// TwinCAT 3 PLC project TAMAR_22mm
// ProgramVersion: 3.1.4023.0
// libraries:
//   Tc2_MC2, * (Beckhoff Automation GmbH)
//   Tc2_Standard, * (Beckhoff Automation GmbH)
//   Tc2_System, * (Beckhoff Automation GmbH)
//   Tc2_Utilities, * (Beckhoff Automation GmbH)
//   Tc3_Module, * (Beckhoff Automation GmbH)
//   VisuDialogs, * (System)
// project tree:
//   Checks/ CheckBounds.TcPOU, CheckDivDInt.TcPOU, CheckDivLInt.TcPOU, CheckDivLReal.TcPOU, CheckDivReal.TcPOU, CheckLRangeSigned.TcPOU, CheckLRangeUnsigned.TcPOU, CheckPointer.TcPOU, CheckRangeSigned.TcPOU, CheckRangeUnsigned.TcPOU
//   DUTs/ ePistonStatus.TcDUT, E_CONVAYOR_STATE.TcDUT, E_EventType.TcDUT (not stored), E_MAIN_STATE.TcDUT, E_PISTON_STATE.TcDUT (not stored), E_PISTON_TYPE.TcDUT (not stored), E_STATION_STATE.TcDUT, ST_CART.TcDUT, ST_CsvTableRowData.TcDUT, ST_Event.TcDUT, ST_PISTON.TcDUT
//   Functions/ F_Linear.TcPOU, UpdateEventTimestampWithSystemTime.TcPOU, UpdateTimeStamp.TcPOU
//   / GlobalTextList.TcGTLO, PlcTask.TcTTO (not stored), Visualization Manager.TcVMO (not stored)
//   GVLs/ GVL.TcGVL, GVL_EVENT_LOGS.TcGVL
//   IO/ EL1809.TcDUT (not stored), EL2869.TcDUT, GVL_IO.TcGVL, ST_VTUG.TcDUT (not stored)
//   POUs/AXES/ FB_Axis.TcPOU
//   POUs/ FB_CART.TcPOU, FB_ERROR_CODE.TcPOU, FB_EventLogger.TcPOU, FB_PISTON.TcPOU, MAIN.TcPOU, MOTORS.TcPOU, PISTONS_CYCLE.TcPOU, prg_CSV_V2.TcPOU
//   POUs/PISTONS/ E_PIST_STATUS.TcDUT, E_PIST_TYPE.TcDUT, FB_PIST.TcPOU, GVL_PIST.TcGVL, PIST_CYCLE.TcPOU
//   STATIONS/ FB_CLEAN.TcPOU, FB_DROP.TcPOU, FB_MAIN_CONV.TcPOU, FB_SEPARATE.TcPOU, FB_STATION.TcPOU, FB_SUPPLY.TcPOU, FB_SUPPLY_CONV.TcPOU, _SEPARATE.TcPOU
// real-time tasks:
//   TASK PlcTask: cycle T#10ms, priority 20, ADS port 350
// motion (NC):
//   TASK NC-Task 1 SAF: cycle T#2ms, priority 4, ADS port 501
//   TASK NC-Task 1 SVB: cycle T#10ms, priority 8, ADS port 511
//   AXIS MAIN (id 1)
//     OtherSettings: AllowMotionCmdToSlave=true
//     encoder EncType=19
//       EncPara: MaxCount=#xffffffff
//     drive DrvType=16
//       DrvPara: MaxCount=#xffffffff, DriveControlDWord=#x00000100
//         Analog: TorqueSetpointScale=10, ScaleFactorActTorque=0.1
//         TimeComp: TaskDelayCycles=1
//     controller CtrType=1
//       CtrPara: PriorControlFactor=1
//         Observer: BandWidth=20
//   AXIS SUPPLY (id 2)
//     OtherSettings: AllowMotionCmdToSlave=true
//     encoder EncType=19
//       EncPara: MaxCount=#xffffffff
//     drive DrvType=16
//       DrvPara: MaxCount=#xffffffff, DriveControlDWord=#x00000100
//         Analog: TorqueSetpointScale=10, ScaleFactorActTorque=0.1
//         TimeComp: TaskDelayCycles=1
//     controller CtrType=1
//       CtrPara: PriorControlFactor=1
//         Observer: BandWidth=20
//   AXIS JACK1 (id 3)
//     OtherSettings: AllowMotionCmdToSlave=true
//     encoder EncType=1
//     drive DrvType=5
//       Analog: TorqueSetpointScale=10, ScaleFactorActTorque=0.1
//       TimeComp: TaskDelayCycles=1
//     controller CtrType=1
//       CtrPara: PriorControlFactor=1
//         Observer: BandWidth=20
//   AXIS JACK2 (id 4)
//     OtherSettings: AllowMotionCmdToSlave=true
//     encoder EncType=1
//     drive DrvType=5
//       Analog: TorqueSetpointScale=10, ScaleFactorActTorque=0.1
//     controller CtrType=1
//       CtrPara: PriorControlFactor=1
//         Observer: BandWidth=20
// I/O:
//   DEVICE Device 3 (EtherCAT), AmsNetId 5.109.70.127.4.1
//     Term 1 (EK1100) [EK1100 EtherCAT Coupler (2A E-Bus)]
//       Term 2 (EL1809) [EL1809 16Ch. Dig. Input 24V, 3ms]
//       Term 10 (EL1809) [EL1809 16Ch. Dig. Input 24V, 3ms]
//       Term 11 (EL1809) [EL1809 16Ch. Dig. Input 24V, 3ms]
//       Term 13 (EL1809) [EL1809 16Ch. Dig. Input 24V, 3ms]
//       Term 3 (EL2869) [EL2869 16Ch. Dig Output 24V, 0.5A, Diagnostic]
//       Term 4 (EL6224) [EL6224 (IO Link Master)]
//       Term 15 (EL9011) [EL9011 End Terminal]
//       Term 7 (EL9011) [EL9011 End Terminal]
//     MAIN
//     SUPPLY [CD02 EtherCAT Drive (CoE)]
// variable links:
//   (this object) <-> Device 3 (EtherCAT)/MAIN
//     Drive/Inputs/In/nDataIn1 <-> TxPDO 1/Following Error Actual Value
//     Drive/Inputs/In/nDataIn3[0] <-> TxPDO 4/Torque Actual Value
//     Drive/Inputs/In/nDcOutputTime <-> InfoData/DcOutputShift
//     Drive/Inputs/In/nState1 <-> TxPDO 4/Statusword
//     Drive/Inputs/In/nState2 <-> TxPDO 4/Statusword @bit 8
//     Drive/Inputs/In/nState4 @bit 1 <-> WcState/InputToggle
//     Drive/Inputs/In/nState4 <-> WcState/WcState
//     Drive/Inputs/In/nState5 <-> TxPDO 3/Modes of Operation Display
//     Drive/Outputs/Out/nCtrl1 <-> RxPDO 4/Controlword
//     Drive/Outputs/Out/nCtrl2 <-> RxPDO 4/Controlword @bit 8
//     Drive/Outputs/Out/nCtrl5 <-> RxPDO 4/Modes of Operation
//     Drive/Outputs/Out/nDataOut1 <-> RxPDO 1/Target Position
//     Drive/Outputs/Out/nDataOut2 <-> RxPDO 2/Target Velocity
//     Drive/Outputs/Out/nDataOut3[0] <-> RxPDO 4/Torque Offset
//     Drive/Outputs/Out/nDataOut4[0] <-> RxPDO 3/Target Torque
//     Enc/Inputs/In/nDataIn1 <-> TxPDO 2/Position Actual Value
//     Enc/Inputs/In/nDcInputTime <-> InfoData/DcInputShift
//     Enc/Inputs/In/nState4 @bit 1 <-> WcState/InputToggle
//     Enc/Inputs/In/nState4 <-> WcState/WcState
//   (this object) <-> Device 3 (EtherCAT)/SUPPLY
//     Drive/Inputs/In/nDataIn1 <-> TxPDO 1/Following Error Actual Value
//     Drive/Inputs/In/nDataIn3[0] <-> TxPDO 4/Torque Actual Value
//     Drive/Inputs/In/nDcOutputTime <-> InfoData/DcOutputShift
//     Drive/Inputs/In/nState1 <-> TxPDO 4/Statusword
//     Drive/Inputs/In/nState2 <-> TxPDO 4/Statusword @bit 8
//     Drive/Inputs/In/nState4 @bit 1 <-> WcState/InputToggle
//     Drive/Inputs/In/nState4 <-> WcState/WcState
//     Drive/Inputs/In/nState5 <-> TxPDO 3/Modes of Operation Display
//     Drive/Outputs/Out/nCtrl1 <-> RxPDO 4/Controlword
//     Drive/Outputs/Out/nCtrl2 <-> RxPDO 4/Controlword @bit 8
//     Drive/Outputs/Out/nCtrl5 <-> RxPDO 4/Modes of Operation
//     Drive/Outputs/Out/nDataOut1 <-> RxPDO 1/Target Position
//     Drive/Outputs/Out/nDataOut2 <-> RxPDO 2/Target Velocity
//     Drive/Outputs/Out/nDataOut3[0] <-> RxPDO 4/Torque Offset
//     Drive/Outputs/Out/nDataOut4[0] <-> RxPDO 3/Target Torque
//     Enc/Inputs/In/nDataIn1 <-> TxPDO 2/Position Actual Value
//     Enc/Inputs/In/nDcInputTime <-> InfoData/DcInputShift
//     Enc/Inputs/In/nState4 @bit 1 <-> WcState/InputToggle
//     Enc/Inputs/In/nState4 <-> WcState/WcState
//   TAMAR_22mm Instance <-> Device 3 (EtherCAT)/Term 1 (EK1100)/Term 2 (EL1809)
//     PlcTask Inputs/GVL_IO.inputs[1]/ch{1..16} <-> Channel {1..16}/ch{1..16}  (16 links)
//   TAMAR_22mm Instance <-> Device 3 (EtherCAT)/Term 1 (EK1100)/Term 3 (EL2869)
//     PlcTask Outputs/GVL_IO.outputs[1]/ch{1..16} <-> DOS Outputs Channel {1..16}/Output  (16 links)
//   TAMAR_22mm Instance <-> Device 3 (EtherCAT)/Term 1 (EK1100)/Term 4 (EL6224)
//     PlcTask Outputs/GVL_IO.uIOLINK1 <-> IO-Link Port1_out/GVL_IO.uIOLINK1
//     PlcTask Outputs/GVL_IO.uIOLINK2 <-> IO-Link Port2_out/GVL_IO.uIOLINK2
//   TAMAR_22mm Instance <-> NC-Task 1 SAF/Axes/JACK1
//     PlcTask Inputs/GVL.Axis_JACK1.Axis.NcToPlc <-> Outputs/ToPlc
//     PlcTask Outputs/GVL.Axis_JACK1.Axis.PlcToNc <-> Inputs/FromPlc
//   TAMAR_22mm Instance <-> NC-Task 1 SAF/Axes/JACK2
//     PlcTask Inputs/GVL.Axis_JACK2.Axis.NcToPlc <-> Outputs/ToPlc
//     PlcTask Outputs/GVL.Axis_JACK2.Axis.PlcToNc <-> Inputs/FromPlc
//   TAMAR_22mm Instance <-> NC-Task 1 SAF/Axes/MAIN
//     PlcTask Inputs/GVL.Axis_MAIN.Axis.NcToPlc <-> Outputs/ToPlc
//     PlcTask Outputs/GVL.Axis_MAIN.Axis.PlcToNc <-> Inputs/FromPlc
//   TAMAR_22mm Instance <-> NC-Task 1 SAF/Axes/SUPPLY
//     PlcTask Inputs/GVL.Axis_SUPPLY.Axis.NcToPlc <-> Outputs/ToPlc
//     PlcTask Outputs/GVL.Axis_SUPPLY.Axis.PlcToNc <-> Inputs/FromPlc

// ---- DUTs/ePistonStatus.TcDUT
{attribute 'qualified_only'}
{attribute 'strict'}
TYPE ePistonStatus :
(
	OPENED:=0,CLOSED,OPENING,CLOSING,ERROR,PAUSE
);
END_TYPE

// ---- DUTs/E_CONVAYOR_STATE.TcDUT
{attribute 'qualified_only'}
{attribute 'strict'}
TYPE E_CONVAYOR_STATE :
(
	uninit,
	idle,
	do_move,
	st1,
	st2,
	st3,
	st4,
	st5,
	done,
	pause,
	error,
	homing,
	estop
);
END_TYPE

// ---- DUTs/E_MAIN_STATE.TcDUT
{attribute 'qualified_only'}
{attribute 'strict'}
TYPE E_MAIN_STATE :
(
	uninit,
	idle,
	do_actions,
	move_next,
	done,
	pause,
	error,
	estop,
	homing,
	safety
);
END_TYPE

// ---- DUTs/E_STATION_STATE.TcDUT
{attribute 'qualified_only'}
{attribute 'strict'}
TYPE E_STATION_STATE :
(
	uninit:=0,
	idle,
	homing,
	do_action1,
	do_action2,
	do_action3,
	do_action4,
	do_action5,
	do_action6,
	do_action7,
	do_action8,
	do_action9,
	do_action10,
	do_action11,
	do_action12,
	do_action13,
	do_action14,
	do_action15,
	done,
	pause,
	error,
	estop
);
END_TYPE

// ---- DUTs/ST_CART.TcDUT
TYPE ST_CART :
STRUCT
	nNAME: STRING;
	posX:INT;
	posY:INT;
	color:INT;
	o_color:INT;
	position: INT;
	
END_STRUCT
END_TYPE

// ---- DUTs/ST_CsvTableRowData.TcDUT
TYPE ST_CsvTableRowData :
STRUCT
	sTimeStamp:STRING;
	sType:STRING;
	sSeverity:STRING;
	sIdentity:STRING;
	sName:STRING;
	sText:STRING;
	sROP:STRING;
	sP_TRANSFER:STRING;
	sP_TAP:STRING;
	sP_CAPSULE:STRING;
	sS_FEED:STRING;
	sS_PRODUCT:STRING;
	sH_FEED:STRING;
	sH_PRODUCT:STRING;
	sSel_FEED:STRING;
	sSel_PRODUCT:STRING;
	sUnit:STRING;
END_STRUCT
END_TYPE

// ---- DUTs/ST_Event.TcDUT
TYPE ST_Event :
STRUCT
	eEventType: E_EventType; 
	eEventSeverity: TcEventSeverity;
	nEventIdentity: UDINT;
	sEventName: STRING(255);
	sEventText: STRING(255);
	dtTimestamp: DATE_AND_TIME;
	
END_STRUCT
END_TYPE

// ---- DUTs/ST_PISTON.TcDUT
 TYPE ST_PISTON :
STRUCT
	ePISTON_TYPE: E_PISTON_TYPE;
	
	nNAME: STRING;
	openTime: REAL:=5;
	closeTime: REAL:=5;
	timeoutOpen:  TIME:=T#5S;
	timeoutClose: TIME:=T#5S;
	bOPEN_BY_DEFAULT: BOOL:= FALSE;
	
	
END_STRUCT
	
END_TYPE

// ---- IO/EL2869.TcDUT
TYPE EL2869 :
STRUCT
	ch1		:BOOL;
	ch2		:BOOL;
	ch3		:BOOL;
	ch4		:BOOL;
	ch5		:BOOL;
	ch6		:BOOL;
	ch7		:BOOL;
	ch8		:BOOL;
	ch9		:BOOL;
	ch10		:BOOL;
	ch11		:BOOL;
	ch12		:BOOL;
	ch13		:BOOL;
	ch14		:BOOL;
	ch15		:BOOL;
	ch16		:BOOL;	
END_STRUCT
END_TYPE

// ---- POUs/PISTONS/E_PIST_STATUS.TcDUT
{attribute 'qualified_only'}
{attribute 'strict'}
TYPE E_PIST_STATUS :
(
	UNINIT:=0,INIT,READY,OPENED,CLOSED,OPENING,CLOSING,ERROR,PAUSE,NEUTRALIZE,NEUTRAL
);
END_TYPE

// ---- POUs/PISTONS/E_PIST_TYPE.TcDUT
{attribute 'qualified_only'}
{attribute 'strict'}
TYPE E_PIST_TYPE :
(
	NO_SENSORS:=0,
	ONLY_OPEN,
	ONLY_CLOSE,
	BOTH
);
END_TYPE

// ---- GVLs/GVL.TcGVL
 //{attribute 'qualified_only'}
VAR_GLOBAL
	{attribute 'OPC.UA.DA' := '1'}
	rVal11:REAL;
	{attribute 'OPC.UA.DA' := '1'}
	rVal2:REAL;
	{attribute 'OPC.UA.DA' := '1'}
	bTest:BOOL;
	
	
	bValve: ARRAY[1..64] OF BOOL;
	//======================================== IO =====================================
	nanlogIn1 AT%I*:INT;
	rAnalogIn:REAL;
	//======================================== stations =============================== 
	supply_station_num: INT:=1;
	separate1_station_num: INT:=5;
	separate2_station_num: INT:=9;
	bullet_check_num: INT:=15;
	dispose_station_num:INT:=15;
	clean_station_num: INT:=23;
	primer_station_num: INT:=27;
	drop_station_num: INT:=33;
	
	total_ready:INT:=0;
	iNUMBER_OF_PISTONS:INT:=22;
	conv_length: INT:=1350;
	conv_height: INT:=290;
	num_of_carts:INT:=18;
	X_OFFSET: INT:=380; 
	Y_OFFSET: INT:=352;
	stPISTON_PARAM: ARRAY[1..22] OF  ST_PISTON;
	//fbPiston: ARRAY[1..22] OF FB_PISTON;
	
	fbCART: ARRAY[1..18] OF FB_CART;
	Axis_MAIN:FB_Axis;
	Axis_SUPPLY:FB_Axis;
	Axis_JACK1:FB_Axis;
	Axis_JACK2:FB_Axis;
	
	posArrX:ARRAY[1..36] OF INT;
	posArrY:ARRAY[1..36] OF INT;
	
	eMAIN_STATE: E_MAIN_STATE:= E_MAIN_STATE.uninit;
	eSUPPLY: E_STATION_STATE:=E_STATION_STATE.uninit;
	eSEPARATE1: E_STATION_STATE:=E_STATION_STATE.uninit;
	eSEPARATE2: E_STATION_STATE:=E_STATION_STATE.uninit;
	e_SEPARATE1: E_STATION_STATE:=E_STATION_STATE.uninit;
	e_SEPARATE2: E_STATION_STATE:=E_STATION_STATE.uninit;
	eCLEAN: E_STATION_STATE:=E_STATION_STATE.uninit;
	eDROP: E_STATION_STATE:=E_STATION_STATE.uninit;
	eMAIN_CONVAYOR_STATE: E_CONVAYOR_STATE:=E_CONVAYOR_STATE.uninit;
	eSUPPLY_CONVAYOR_STATE: E_CONVAYOR_STATE:=E_CONVAYOR_STATE.uninit;
	
	bSTART: BOOL:=FALSE;// start main state machine
	sup_RUNNING: BOOL:=FALSE;// supply id runing
	clean_RUNNING: BOOL:=FALSE;// cleaning runing
	bS1_RUNNING: BOOL:=FALSE; // station 1 is running
	bS2_RUNNING: BOOL:=FALSE; // station 2 is running
	bCONV_MAIN_INPOS: BOOL:=FALSE; // convayor in position
	bCONV_SUPPLY_INPOS: BOOL:=FALSE; // convayor in position
	bPAUSE_MAIN: BOOL:=FALSE;
	bINIT_MAIN: BOOL:=FALSE;
	b_E_STOP:BOOL:=FALSE;
	b_RESET:BOOL:=FALSE;
	bSafety_error:BOOL:=FALSE;
	b_sense_home1: BOOL:=TRUE;
	b_sense_home2: BOOL;
	b_sense_home3: BOOL:=TRUE;
	bManual_Mode:BOOL:=FALSE;
	bBulletSensor:BOOL:=FALSE;
END_VAR

// ---- GVLs/GVL_EVENT_LOGS.TcGVL
//{attribute 'qualified_only'}
VAR_GLOBAL
	// ================================== error and logs ==============================
	sError:STRING;
	gEventType: STRING(255); 
	gEventSeverity: STRING(255);
	gEventIdentity: UDINT:=0;
	gEventText: STRING(255):='Startup Event';
	gEventName: STRING(255);
	sEventTime: STRING(255);
	fbEventLogger: FB_EventLogger;
	WriteLogToFile:BOOL:=FALSE;
	sLog:STRING(255);
	bBuffer_full:BOOL:=FALSE;
END_VAR

// ---- IO/GVL_IO.TcGVL
//{attribute 'qualified_only'}
VAR_GLOBAL
	uIOLINK1 AT%Q* : ULINT;
	uIOLINK2 AT%Q* : ULINT;	

	inputs AT %I* : ARRAY [1..4] OF EL1809;
	outputs AT %Q* : ARRAY[1..2] OF EL2869;
	
	//manifold AT %Q* : ARRAY[1..3] OF ST_VTUG;

END_VAR

// ---- POUs/PISTONS/GVL_PIST.TcGVL
//{attribute 'qualified_only'}
VAR_GLOBAL
	fbPist:  ARRAY[1..31] OF FB_PIST;
END_VAR

// ---- POUs/FB_PISTON.TcPOU
FUNCTION_BLOCK FB_PISTON

VAR_INPUT
	stPISTON:   REFERENCE TO ST_PISTON;
	bDepened_open1:BOOL:=TRUE;
	bDepened_open2:BOOL:=TRUE;
	bDepened_close1:BOOL:=TRUE;
	bDepened_close2:BOOL:=TRUE;
END_VAR

VAR_OUTPUT
	PistonStatus:ePistonStatus;
	bVALVE_OPEN: BOOL;
	bVALVE_CLOSE: BOOL;
END_VAR

VAR
	bMANUAL:BOOL:=FALSE;
	sName:STRING;
	bCMD_OPEN_SWR: BOOL;
	bCMD_CLOSE_SWR: BOOL;
	bCMD_OPEN: BOOL;
	bSEN_OPEN AT%I*: BOOL;
	bSEN_CLOSE AT%I*: BOOL;
	timerOpening:ton;
	timerClosing:ton;
	timeoutOpening:ton;
	timeoutClosing:ton;
	bSTARTUP: BOOL:=FALSE;
	rtrigMANUAL: R_TRIG;
	rtrig_OPEN_ERROR: R_TRIG;
	rtrig_CLOSE_ERROR: R_TRIG;
	rtrig_OPEN_CONDITION: R_TRIG;
	rtrig_CLOSE_CONDITION: R_TRIG;
	bERROR:BOOL:=FALSE;
	
	bError_Condition_open:BOOL;
	bError_Condition_close:BOOL;
END_VAR



IF NOT bSTARTUP THEN
	bCMD_OPEN:=stPISTON.bOPEN_BY_DEFAULT;
	bSTARTUP:=TRUE;
	sName:=stPISTON.nNAME;
END_IF

rtrigMANUAL(CLK:= bMANUAL, Q=> );
IF rtrigMANUAL.Q THEN
	bCMD_OPEN:=bCMD_OPEN_SWR;
END_IF
// opening error timeout  triger
rtrig_OPEN_ERROR(CLK:=(timeoutOpening.Q AND (stPISTON.ePISTON_TYPE = E_PISTON_TYPE.ONLY_OPEN OR stPISTON.ePISTON_TYPE = E_PISTON_TYPE.BOTH)), Q=> );
IF rtrig_OPEN_ERROR.Q THEN
	PistonStatus:=ePistonStatus.ERROR;
	gEventText:='PISTON OPENING TIMEOUT:';
	A_OPEN_ERROR();
END_IF
// closing error timeout triger
rtrig_CLOSE_ERROR(CLK:=(timeoutClosing.Q AND (stPISTON.ePISTON_TYPE = E_PISTON_TYPE.ONLY_CLOSE OR stPISTON.ePISTON_TYPE = E_PISTON_TYPE.BOTH)), Q=> );
IF rtrig_CLOSE_ERROR.Q THEN
	PistonStatus:=ePistonStatus.ERROR;
	gEventText:='PISTON CLOSING TIMEOUT:';
	A_CLOSE_ERROR();
END_IF
//opening condition error triger
rtrig_OPEN_CONDITION(CLK:=bError_Condition_open, Q=> );
IF rtrig_OPEN_CONDITION.Q THEN
	PistonStatus:=ePistonStatus.ERROR;
	gEventText:='PISTON OPENING CONDITION:';
	A_OPEN_ERROR();
END_IF
//closing condition error triger
rtrig_CLOSE_CONDITION(CLK:=bError_Condition_close, Q=> );
IF rtrig_CLOSE_CONDITION.Q THEN
	PistonStatus:=ePistonStatus.ERROR;
	gEventText:='PISTON CLOSING CONDITION:';
	A_CLOSE_ERROR();
END_IF


timerOpening(IN:= bVALVE_OPEN, PT:=REAL_TO_TIME(stPISTON.openTime*1000) , Q=> , ET=> );
timerClosing(IN:= NOT bVALVE_OPEN, PT:=REAL_TO_TIME(stPISTON.closeTime*1000) , Q=> , ET=> );
timeoutOpening(IN:= bVALVE_OPEN AND NOT bSEN_OPEN, PT:= stPISTON.timeoutOpen, Q=> , ET=> );
timeoutClosing(IN:= NOT bVALVE_OPEN AND NOT bSEN_CLOSE, PT:= stPISTON.timeoutClose, Q=> , ET=> );

IF bMANUAL THEN
	IF bCMD_OPEN AND bDepened_open1 THEN
		bVALVE_OPEN:= bCMD_OPEN;
		bError_Condition_open:=FALSE;	
	ELSIF bCMD_OPEN AND NOT bDepened_open1 THEN
		bError_Condition_open:=TRUE; 
		//gEventText:='PISTON OPENING CONDITION:';
		//A_OPEN_ERROR();
	END_IF
	
	IF NOT bCMD_OPEN AND bDepened_close1 THEN
		bVALVE_OPEN:= bCMD_OPEN;
		bError_Condition_close:=FALSE;	
	ELSIF NOT bCMD_OPEN AND NOT bDepened_close1 THEN
		bError_Condition_close:=TRUE;
		//gEventText:='PISTON CLOSING CONDITION:';
		//A_CLOSE_ERROR();
	END_IF
	
ELSE
	IF bCMD_OPEN_SWR AND bDepened_open1 THEN
		bVALVE_OPEN:= bCMD_OPEN_SWR;
		bError_Condition_open:=FALSE;	
	ELSIF bCMD_OPEN_SWR AND NOT bDepened_open1 THEN
		bError_Condition_open:=TRUE;
		//gEventText:='PISTON OPENING CONDITION:';
		//A_OPEN_ERROR();
	END_IF
	
	IF NOT bCMD_OPEN_SWR AND bDepened_close1 THEN
		bVALVE_OPEN:= bCMD_OPEN_SWR;
		bError_Condition_close:=FALSE;	
	ELSIF NOT bCMD_OPEN_SWR AND NOT bDepened_close1 THEN
		bError_Condition_close:=TRUE;
		//gEventText:='PISTON CLOSING CONDITION:';
		//A_CLOSE_ERROR();
	END_IF
END_IF
bVALVE_CLOSE:=NOT bVALVE_OPEN;


CASE stPISTON.ePISTON_TYPE OF
	0://NO_SENSORS
		IF bVALVE_OPEN AND NOT timerOpening.Q THEN
			PistonStatus:=ePistonStatus.OPENING;
		ELSIF bVALVE_OPEN AND timerOpening.Q THEN
			PistonStatus:=ePistonStatus.OPENED;
		ELSIF bVALVE_CLOSE AND NOT timerClosing.Q THEN
			PistonStatus:=ePistonStatus.CLOSING;
		ELSIF bVALVE_CLOSE AND timerClosing.Q THEN
			PistonStatus:=ePistonStatus.CLOSED;
		END_IF
		
 
	
	1://only open sensor
	
		IF bVALVE_OPEN AND NOT bSEN_OPEN AND NOT timeoutOpening.Q THEN
			PistonStatus:=ePistonStatus.OPENING;
		ELSIF bVALVE_OPEN AND bSEN_OPEN THEN
			PistonStatus:=ePistonStatus.OPENED;
		ELSIF bVALVE_CLOSE AND NOT timerClosing.Q THEN
			PistonStatus:=ePistonStatus.CLOSING;
		ELSIF bVALVE_CLOSE AND timerClosing.Q THEN
			PistonStatus:=ePistonStatus.CLOSED;
		END_IF
	
	2:// only close sensor
		IF bVALVE_OPEN AND NOT timerOpening.Q THEN
			PistonStatus:=ePistonStatus.OPENING;
		ELSIF bVALVE_OPEN AND timerOpening.Q THEN
			PistonStatus:=ePistonStatus.OPENED;
		ELSIF bVALVE_CLOSE AND NOT bSEN_CLOSE AND NOT timeoutClosing.Q THEN
			PistonStatus:=ePistonStatus.CLOSING;
		ELSIF bVALVE_CLOSE AND bSEN_CLOSE THEN
			PistonStatus:=ePistonStatus.CLOSED;
		END_IF
	
	
	3://both sensors
		IF bVALVE_OPEN AND NOT bSEN_OPEN AND NOT timeoutOpening.Q THEN
			PistonStatus:=ePistonStatus.OPENING;
		ELSIF bVALVE_OPEN AND bSEN_OPEN THEN
			PistonStatus:=ePistonStatus.OPENED;
		ELSIF bVALVE_CLOSE AND NOT bSEN_CLOSE AND NOT timeoutClosing.Q THEN
			PistonStatus:=ePistonStatus.CLOSING;
		ELSIF bVALVE_CLOSE AND bSEN_CLOSE THEN
			PistonStatus:=ePistonStatus.CLOSED;
		END_IF
	
END_CASE

//IF timeoutOpening.Q AND (stPISTON.ePISTON_TYPE = E_PISTON_TYPE.ONLY_OPEN OR stPISTON.ePISTON_TYPE = E_PISTON_TYPE.BOTH)  THEN
//	PistonStatus:=ePistonStatus.ERROR;
//	A_OPEN_ERROR();
//END_IF
//IF timeoutClosing.Q  AND (stPISTON.ePISTON_TYPE = E_PISTON_TYPE.ONLY_CLOSE OR stPISTON.ePISTON_TYPE = E_PISTON_TYPE.BOTH)  THEN
//	PistonStatus:=ePistonStatus.ERROR;
//	A_CLOSE_ERROR();
//END_IF

ACTION A_CLOSE:
bCMD_OPEN_SWR:=FALSE;
END_ACTION

ACTION A_CLOSE_ERROR:
gEventType:= 'Alarm'; 
gEventSeverity:= 'Error';
gEventIdentity:=1002;
gEventName:= stPISTON.nNAME;
fbEventLogger.mAdd();
END_ACTION

ACTION A_DEFAULT:

IF stPISTON.bOPEN_BY_DEFAULT THEN
	bCMD_OPEN_SWR:=TRUE;
ELSE
	bCMD_OPEN_SWR:=FALSE;
END_IF
END_ACTION

ACTION A_OPEN:
bCMD_OPEN_SWR:=TRUE;
END_ACTION

ACTION A_OPEN_ERROR:
gEventType:= 'Alarm'; 
gEventSeverity:= 'Error';
gEventIdentity:=1001;
gEventName:= stPISTON.nNAME;
fbEventLogger.mAdd();
END_ACTION

END_FUNCTION_BLOCK

// ---- POUs/FB_CART.TcPOU
FUNCTION_BLOCK FB_CART
VAR_INPUT
	stCART: ST_CART;
END_VAR
VAR_OUTPUT
	
END_VAR

VAR
	inner_counter: INT;
END_VAR

ACTION A_CHECK:
IF stCART.position = bullet_check_num THEN
		IF bBulletSensor THEN
			stCART.color:=89;
			bSafety_error:=TRUE;
			b_E_STOP:=TRUE;
				
			gEventType:= 'Alarm'; 
			gEventSeverity:= 'Safety';
			gEventIdentity:=9001;
			gEventName:= stCART.nNAME;
			gEventText:='BULLETS NOT PICKED:';
			fbEventLogger.mAdd();
		END_IF
	END_IF
END_ACTION

ACTION A_STEP:
IF stCART.position < num_of_carts*2 THEN
	


	IF stCART.position = supply_station_num THEN
		IF NOT MAIN.fbSUPPLY.bSkip THEN
			stCART.color:=2;
		ELSE
			stCART.color:=99;
		END_IF
		stCART.o_color:=2;
	END_IF  
	IF stCART.position = separate1_station_num THEN
		IF NOT MAIN.fbSEPARATION1.bSkip THEN
			IF stCART.color = 2 THEN
				stCART.color:=3;
			END_IF
		ELSE
			stCART.color:=99;
		END_IF
		stCART.o_color:=3;
		
	END_IF 
	IF stCART.position = separate2_station_num THEN
		IF NOT MAIN.fbSEPARATION2.bSkip THEN
			IF stCART.color = 3 THEN
				stCART.color:=4;
			END_IF
		ELSE
			stCART.color:=99;
		END_IF
		stCART.o_color:=4;
	END_IF 
	
	
	
	IF stCART.position = clean_station_num THEN
		IF NOT MAIN.fbCLEAN.bSkip THEN
			IF stCART.color = 4 THEN
				stCART.color:=1;
			END_IF
		ELSE
			stCART.color:=99;
		END_IF
		stCART.o_color:=1;
	END_IF 
	
	
	
	stCART.position:= stCART.position+1;
	stCART.posX:=posArrX[stCART.position];
	stCART.posY:=posArrY[stCART.position];
ELSE
	stCART.position:= 1;
	stCART.posX:=posArrX[stCART.position];
	stCART.posY:=posArrY[stCART.position];
	
END_IF
END_ACTION

END_FUNCTION_BLOCK

// ---- POUs/MAIN.TcPOU
PROGRAM MAIN
VAR
	counter1:INT:=0;
	counter:INT:=0;
	iNUMBER1 : INT:=2;
	sNAME1 : STRING(255):='23_5A';
	Trigger : BOOL;
	rtrigRESET: R_TRIG;
	rtrigE_STOP: R_TRIG;
	rtrigSTART: R_TRIG;
	rtrigPAUSE: R_TRIG;
	rtrigINIT: R_TRIG;
	ftrigRERUN: F_TRIG;
	temp_state:E_MAIN_STATE;
	temp_supply_state:E_STATION_STATE;
	temp_sep1_state:E_STATION_STATE;
	temp_sep2_state:E_STATION_STATE;
	temp_clean_state:E_STATION_STATE;
	temp_drop_state:E_STATION_STATE;
	temp_conv_state:E_CONVAYOR_STATE;
	temp_supconv_state:E_CONVAYOR_STATE;
	bHomed:BOOL:=FALSE;
	fbSEPARATION1: FB_SEPARATE;		
	fbSEPARATION2: FB_SEPARATE;	
	fb_SEPARATE1: _SEPARATE;
	fb_SEPARATE2: _SEPARATE;
	fbCLEAN: FB_CLEAN;
	fbDROP: FB_DROP;
	fbSUPPLY: FB_SUPPLY;
	fbMAIN_CONV: FB_MAIN_CONV;
	fbSUPPLY_CONV: FB_SUPPLY_CONV;
	
	
	
	action_timeout: TON:=(PT:=T#20S); 
	move_timeout: TON;
	bTIMEOUT:BOOL:=FALSE;
	
	bFirstRun:BOOL:=TRUE;
END_VAR

IF bFirstRun THEN
	fbEventLogger.mAdd();
	bFirstRun:=FALSE;
END_IF

//uIOLINK1.10:=1;
//uIOLINK1.11:=1;

rAnalogIn:=F_Linear(nanlogIn1,200,31170,0,2000);
//PISTONS_CYCLE();
A_PISTON_ERROR_CHECK();
fbMAIN_CONV(fbAxis:=Axis_MAIN);
fbSUPPLY_CONV(fbAxis:=Axis_SUPPLY);

fb_SEPARATE1(piston_updown:=  fbPist[12],
			  piston_colet1:=  fbPist[14],
			   piston_colet2:=  fbPist[15],
			    piston_colet3:=  fbPist[16],
				 piston_colet4:=  fbPist[30],
			  piston_tray:=  fbPist[17],
			  piston_pins:=  fbPist[13],
			  piston_tray_door:=  fbPist[19],
			  piston_tray_push:=  fbPist[18],
			  eState:= e_SEPARATE1,
			  fbAxis:=Axis_JACK1,
			  station_num:=separate1_station_num);
	

fb_SEPARATE2(piston_updown:=  fbPist[20],
			  piston_colet1:=  fbPist[22],
			   piston_colet2:=  fbPist[23],
			    piston_colet3:=  fbPist[24],
				 piston_colet4:=  fbPist[25],
			  piston_tray:=  fbPist[26],
			  piston_pins:=  fbPist[21],
			   piston_tray_door:=  fbPist[28],
			  piston_tray_push:=  fbPist[27],
			  eState:= e_SEPARATE2,
			  fbAxis:=Axis_JACK2,
 			  station_num:=separate2_station_num);			  

	
fbCLEAN(pClean:=  fbPist[6]);
fbDROP(pPush:=  fbPist[9],pOpen1:=  fbPist[10],pOpen2:=  fbPist[11]);
fbSUPPLY(pPush:=fbPist[1],pLock1:=fbPist[2],pLock2:=fbPist[3],pOpen1:=fbPist[4],pOpen2:=fbPist[5]);
prg_CSV_V2();
MOTORS();
PIST_CYCLE();
rtrigRESET(CLK:= b_RESET, Q=> );
rtrigE_STOP(CLK:= b_E_STOP, Q=> );
rtrigINIT(CLK:= bINIT_MAIN, Q=> );
rtrigSTART(CLK:= bSTART, Q=> );
rtrigPAUSE(CLK:= bPAUSE_MAIN, Q=> );
ftrigRERUN(CLK:= bPAUSE_MAIN, Q=> );
action_timeout(IN:=bTIMEOUT);

//MAIN_STATE_MACHINE:
CASE eMAIN_STATE OF
	E_MAIN_STATE.homing:   // homing fo all stations
		eSUPPLY := E_STATION_STATE.homing;
		e_SEPARATE1 := E_STATION_STATE.homing;
		e_SEPARATE2 := E_STATION_STATE.homing;
		eCLEAN := E_STATION_STATE.homing;
		eDROP := E_STATION_STATE.homing;
		eMAIN_CONVAYOR_STATE := E_CONVAYOR_STATE.homing;
		eSUPPLY_CONVAYOR_STATE:=E_CONVAYOR_STATE.homing;
		//IF fbSEPARATION1.bHomed AND fbSEPARATION2.bHomed THEN
			eMAIN_STATE:=E_MAIN_STATE.idle;
			bHomed:=TRUE;
		//END_IF
		
	E_MAIN_STATE.uninit:
		IF NOT bHomed THEN
			eMAIN_STATE:=E_MAIN_STATE.homing;
		ELSE
			bTIMEOUT:=FALSE;
			bPAUSE_MAIN:=FALSE;
			eSUPPLY := E_STATION_STATE.unInit;
			//eSEPARATE1 := E_STATION_STATE.unInit;
			e_SEPARATE1 := E_STATION_STATE.unInit;
			e_SEPARATE2 := E_STATION_STATE.unInit;
			eCLEAN := E_STATION_STATE.unInit;
			eDROP := E_STATION_STATE.unInit;
			eMAIN_CONVAYOR_STATE := E_CONVAYOR_STATE.unInit;
			eSUPPLY_CONVAYOR_STATE:=E_CONVAYOR_STATE.unInit;
			eMAIN_STATE:=E_MAIN_STATE.idle;
		END_IF
		
		
		
	E_MAIN_STATE.idle:
		IF rtrigSTART.Q THEN
			IF b_sense_home1 AND NOT b_sense_home2 AND b_sense_home3 THEN 
				eMAIN_STATE:=E_MAIN_STATE.safety;
			END_IF
		END_IF
	
	E_MAIN_STATE.safety:
		A_SAFETY_CHECK();
		IF NOT b_E_STOP THEN
			eMAIN_STATE:=E_MAIN_STATE.do_actions;
		ELSE
			eMAIN_STATE:=E_MAIN_STATE.estop;
		END_IF
	
	E_MAIN_STATE.do_actions:
		bTIMEOUT:=TRUE;
		IF b_sense_home1 AND NOT b_sense_home2 AND b_sense_home3 THEN 
			IF eSUPPLY = E_STATION_STATE.idle THEN     
				eSUPPLY := E_STATION_STATE.do_action1;
			END_IF
			IF e_SEPARATE1 = E_STATION_STATE.idle THEN
				e_SEPARATE1 := E_STATION_STATE.do_action1;
			END_IF
			IF e_SEPARATE2 = E_STATION_STATE.idle THEN
				e_SEPARATE2 := E_STATION_STATE.do_action1;
			END_IF
			IF eCLEAN = E_STATION_STATE.idle THEN
				eCLEAN := E_STATION_STATE.do_action1;
			END_IF
			IF eDROP = E_STATION_STATE.idle THEN
				eDROP := E_STATION_STATE.do_action1;
			END_IF
		END_IF
		IF (e_SEPARATE1 = E_STATION_STATE.done AND e_SEPARATE2 = E_STATION_STATE.done AND eSUPPLY = E_STATION_STATE.done  AND eCLEAN = E_STATION_STATE.done AND eDROP = E_STATION_STATE.done) THEN
			eSUPPLY := E_STATION_STATE.idle;
			e_SEPARATE1 := E_STATION_STATE.idle;
			e_SEPARATE2 := E_STATION_STATE.idle;
			eCLEAN := E_STATION_STATE.idle;
			eDROP := E_STATION_STATE.idle;
			eMAIN_STATE:=E_MAIN_STATE.move_next;
			bTIMEOUT:=FALSE;
		END_IF
		
		IF action_timeout.Q THEN
			eMAIN_STATE:=E_MAIN_STATE.error;
		END_IF
		
	E_MAIN_STATE.move_next: 
		IF eMAIN_CONVAYOR_STATE = E_CONVAYOR_STATE.idle THEN
			eMAIN_CONVAYOR_STATE := E_CONVAYOR_STATE.do_move;
		END_IF
		IF eSUPPLY_CONVAYOR_STATE = E_CONVAYOR_STATE.idle THEN
			eSUPPLY_CONVAYOR_STATE := E_CONVAYOR_STATE.do_move;
		END_IF
		IF eMAIN_CONVAYOR_STATE = E_CONVAYOR_STATE.done AND eSUPPLY_CONVAYOR_STATE = E_CONVAYOR_STATE.done THEN
			eMAIN_CONVAYOR_STATE := E_CONVAYOR_STATE.idle;
			eSUPPLY_CONVAYOR_STATE := E_CONVAYOR_STATE.idle;
			eMAIN_STATE:=E_MAIN_STATE.safety;
		END_IF
		
	E_MAIN_STATE.pause: 
		bTIMEOUT:=FALSE;
		IF ftrigRERUN.Q THEN
			eMAIN_STATE:=temp_state;
			eSUPPLY:=temp_supply_state;
			e_SEPARATE1:=temp_sep1_state;
			e_SEPARATE2:=temp_sep2_state;
			eCLEAN:=temp_clean_state;
			eDROP:=temp_drop_state;
			eMAIN_CONVAYOR_STATE:=temp_conv_state;
			eSUPPLY_CONVAYOR_STATE:=temp_conv_state;
		END_IF
		
	E_MAIN_STATE.estop: 
		//estop
	
	E_MAIN_STATE.error:
		// error	

END_CASE

IF rtrigRESET.Q THEN
	fbMAIN_CONV.A_set_cart_spaces();
	fbMAIN_CONV.A_SETUP();
	eMAIN_STATE:=E_MAIN_STATE.uninit;
END_IF

IF rtrigE_STOP.Q THEN
	
	A_ESTOP();
	
END_IF

IF rtrigINIT.Q THEN
	
	//eMAIN_CONVAYOR_STATE := E_CONVAYOR_STATE.estop;
	//eSUPPLY_CONVAYOR_STATE:=E_CONVAYOR_STATE.estop;
	b_E_STOP:=FALSE;
	bSafety_error:=FALSE;
	eMAIN_STATE:=E_MAIN_STATE.uninit;
END_IF

IF rtrigPAUSE.Q THEN
	temp_state:=eMAIN_STATE;
	temp_supply_state:=eSUPPLY;
	temp_sep1_state:=e_SEPARATE1;
	temp_sep2_state:=e_SEPARATE2;
	temp_clean_state:=eCLEAN;
	temp_drop_state:=eDROP;
	temp_conv_state:=eMAIN_CONVAYOR_STATE;
	temp_supconv_state:=eSUPPLY_CONVAYOR_STATE;
	eMAIN_STATE:=E_MAIN_STATE.pause;
	eSUPPLY:=E_STATION_STATE.pause;
	e_SEPARATE1:=E_STATION_STATE.pause;
	e_SEPARATE2:=E_STATION_STATE.pause;
	eMAIN_CONVAYOR_STATE:=E_CONVAYOR_STATE.pause;
	eSUPPLY_CONVAYOR_STATE:=E_CONVAYOR_STATE.pause;
	eCLEAN:=E_STATION_STATE.pause;
	eDROP:=E_STATION_STATE.pause;
	
END_IF

ACTION A_ESTOP:
gEventType:= 'Message'; 
	eMAIN_STATE:=E_MAIN_STATE.estop;
	eSUPPLY := E_STATION_STATE.estop;
	eSEPARATE1 := E_STATION_STATE.estop;
	eSEPARATE2 := E_STATION_STATE.estop;
	eCLEAN := E_STATION_STATE.estop;
	eDROP := E_STATION_STATE.estop;
	eMAIN_CONVAYOR_STATE := E_CONVAYOR_STATE.estop;
	eSUPPLY_CONVAYOR_STATE:=E_CONVAYOR_STATE.estop;
	Axis_MAIN.bHalt:=TRUE;
	Axis_SUPPLY.bHalt:=TRUE;	

	gEventSeverity:= 'Info';
	gEventIdentity:=999;
	gEventName:='MAIN';
	gEventText:='Emergency Stop';
	fbEventLogger.mAdd();
END_ACTION

ACTION A_PISTON_ERROR_CHECK:
FOR counter:=1 TO iNUMBER_OF_PISTONS BY 1 DO
	IF fbPist[counter].PistStatus = E_PIST_STATUS.ERROR THEN
		eMAIN_STATE:=E_MAIN_STATE.error;
		
	END_IF
	
END_FOR;
END_ACTION

ACTION A_SAFETY_CHECK:
FOR counter1:=1 TO num_of_carts BY 1 DO
	fbCART[counter1].A_CHECK();
END_FOR;
END_ACTION

END_PROGRAM

// ---- STATIONS/FB_SEPARATE.TcPOU
FUNCTION_BLOCK FB_SEPARATE EXTENDS FB_STATION
VAR_INPUT
	b_BULL_SENSOR:BOOL:=FALSE;
	piston_updown: REFERENCE TO FB_PIST;
	piston_colet1: REFERENCE TO FB_PIST;
	piston_colet2: REFERENCE TO FB_PIST;
	piston_colet3: REFERENCE TO FB_PIST;
	piston_colet4: REFERENCE TO FB_PIST;
	piston_puller: REFERENCE TO FB_PIST;
	piston_tray: REFERENCE TO FB_PIST;
	piston_pins: REFERENCE TO FB_PIST;
	piston_tray_door: REFERENCE TO FB_PIST;
	piston_tray_push: REFERENCE TO FB_PIST;
	
	
END_VAR
VAR_OUTPUT
	bRUNNING:BOOL :=FALSE;
	bError:BOOL:=FALSE;
END_VAR
VAR
	
	tDelay: TON;
	bDELAY: BOOL:=FALSE;
	E: INT;
	
END_VAR

 tDelay(IN:=bDELAY);

CASE eState OF
	
	E_STATION_STATE.homing:
		piston_updown.A_INIT();
		piston_colet1.A_INIT(); piston_colet2.A_INIT();piston_colet3.A_INIT();piston_colet4.A_INIT();
		piston_tray.A_INIT();
		piston_tray_push.A_INIT();
		piston_tray_door.A_INIT();
		piston_pins.A_INIT();
		eState:= E_STATION_STATE.idle;
		bHomed:=TRUE;
		bError:=FALSE;
		
	E_STATION_STATE.uninit:
		eState:= E_STATION_STATE.homing;

	E_STATION_STATE.idle:
		bRUNNING:=FALSE;
		
	E_STATION_STATE.do_action1://delay and lower device
		IF NOT bSkip THEN
			piston_updown.A_OPEN();
			eState:=E_STATION_STATE.do_action2;
		ELSE
			eState:=E_STATION_STATE.done;
		END_IF
		
	E_STATION_STATE.do_action2:
		
		IF piston_updown.PistStatus= E_PIST_STATUS.OPENED THEN
			piston_colet1.A_OPEN();
			eState:=E_STATION_STATE.do_action3;
		END_IF
	
	E_STATION_STATE.do_action3:
		IF piston_colet1.PistStatus= E_PIST_STATUS.OPENED  THEN
			piston_updown.A_CLOSE();
			piston_tray.A_OPEN();
			eState:=E_STATION_STATE.do_action4;
		END_IF
	
	E_STATION_STATE.do_action4:
		IF TRUE THEN
			piston_colet1.A_CLOSE();
			piston_tray.A_OPEN();
			eState:=E_STATION_STATE.do_action5;
		END_IF
	 
	E_STATION_STATE.do_action5:
		IF piston_tray.PistStatus= E_PIST_STATUS.OPENED AND piston_colet1.PistStatus= E_PIST_STATUS.CLOSED AND piston_updown.PistStatus= E_PIST_STATUS.CLOSED  THEN
			piston_pins.A_OPEN();
			eState:=E_STATION_STATE.do_action6;
		END_IF

	E_STATION_STATE.do_action6:
		IF piston_pins.PistStatus= E_PIST_STATUS.OPENED THEN
			piston_tray_push.A_OPEN();
			piston_tray_door.A_OPEN();
			eState:=E_STATION_STATE.do_action7;
		END_IF
	
	E_STATION_STATE.do_action7:
		IF piston_tray_push.PistStatus= E_PIST_STATUS.OPENED AND piston_tray_door.PistStatus= E_PIST_STATUS.OPENED  THEN
			piston_tray_push.A_CLOSE();
			piston_tray_door.A_CLOSE();
			eState:=E_STATION_STATE.do_action8;
		END_IF	
		
	E_STATION_STATE.do_action8:
		IF piston_tray_push.PistStatus= E_PIST_STATUS.CLOSED AND piston_tray_door.PistStatus= E_PIST_STATUS.CLOSED  THEN
			piston_tray.A_CLOSE();
			piston_pins.A_CLOSE();
			eState:=E_STATION_STATE.do_action9;
		END_IF
			
	E_STATION_STATE.do_action9:
		
		IF piston_tray.PistStatus= E_PIST_STATUS.CLOSED  THEN
			eState:=E_STATION_STATE.done;
		END_IF	
		
	E_STATION_STATE.done:
		bRUNNING:=FALSE;
		bDone:=TRUE;	
		
	E_STATION_STATE.pause:
		//paused

END_CASE

END_FUNCTION_BLOCK

// ---- STATIONS/FB_STATION.TcPOU
FUNCTION_BLOCK FB_STATION
VAR_INPUT
	bSkip:BOOL:=FALSE;
	station_num:INT;
	sName:STRING;
	bFirstRun:BOOL:=FALSE;
	eState: REFERENCE TO  E_STATION_STATE;
	bE_STOP:BOOL:=FALSE;
	bDone:BOOL;
	
END_VAR
VAR_OUTPUT
	bHomed: BOOL:=FALSE;
END_VAR
VAR
END_VAR

END_FUNCTION_BLOCK

// ---- POUs/PISTONS/FB_PIST.TcPOU
FUNCTION_BLOCK FB_PIST
VAR_INPUT
	bNeutral: BOOL:=FALSE;
	bCMD_OPEN: BOOL;
	bMANUAL: BOOL:=FALSE;
	bSEN_OPEN: BOOL;
	bSEN_CLOSE: BOOL;
	bInit: BOOL:=FALSE;
	open_time: TIME;
	close_time: TIME;
	open_timeout:TIME;
	close_timeout:TIME;
	eType: E_PIST_TYPE;
	bDefaultState: BOOL;
	bDepened_open1:BOOL:=TRUE;
	bDepened_open2:BOOL:=TRUE;
	bDepened_close1:BOOL:=TRUE;
	bDepened_close2:BOOL:=TRUE;
	sName:STRING;
END_VAR
VAR_OUTPUT
	pistStatus:E_PIST_STATUS:=E_PIST_STATUS.UNINIT ;
	bVALVE_OPEN: BOOL;
	bVALVE_CLOSE: BOOL;
	bError_Condition_open:BOOL;
	bError_Condition_close:BOOL;
	bERROR:BOOL:=FALSE;
END_VAR
VAR
	
	
	bCMD_OPEN_SWR: BOOL;
	bCMD_CLOSE_SWR: BOOL;
	
	bSTARTUP: BOOL:=FALSE;
	
	bStepDone: BOOL;
END_VAR

IF NOT bSTARTUP THEN
	bCMD_OPEN:=bDefaultState;
	bCMD_OPEN_SWR:=bDefaultState;
	bSTARTUP:=TRUE;
END_IF

IF NOT bMANUAL THEN
	bCMD_OPEN:=bCMD_OPEN_SWR;
END_IF

CASE pistStatus OF
	E_PIST_STATUS.UNINIT:
	IF bInit THEN
		pistStatus:=E_PIST_STATUS.INIT;
	END_IF
	
	E_PIST_STATUS.INIT:
	//
	
	
	IF bCMD_OPEN THEN
		SFCReset:=FALSE;
		pistStatus:=E_PIST_STATUS.OPENING;
	ELSE
		SFCReset:=FALSE;
		pistStatus:=E_PIST_STATUS.CLOSING;
	END_IF
	
	E_PIST_STATUS.NEUTRALIZE:
		bVALVE_CLOSE:=FALSE;
		bVALVE_OPEN :=FALSE;
		pistStatus:=E_PIST_STATUS.NEUTRAL;
		
	E_PIST_STATUS.OPENING:
		open_pist();
		
	E_PIST_STATUS.CLOSING:
		close_pist();
	
	
	E_PIST_STATUS.OPENED:	
	IF NOT bNeutral THEN
		IF NOT bCMD_OPEN THEN
			pistStatus:=E_PIST_STATUS.CLOSING;
		END_IF
	ELSE
		SFCReset:=FALSE;
		pistStatus:=E_PIST_STATUS.NEUTRALIZE;
	END_IF
	
	E_PIST_STATUS.CLOSED:	
	IF NOT bNeutral THEN
		IF bCMD_OPEN THEN
			pistStatus:=E_PIST_STATUS.OPENING;
		END_IF
	ELSE
		SFCReset:=FALSE;
		pistStatus:=E_PIST_STATUS.NEUTRALIZE;
	END_IF
	
	E_PIST_STATUS.NEUTRAL:	
	IF NOT bNeutral THEN
		IF bCMD_OPEN THEN
			SFCReset:=FALSE;
			pistStatus:=E_PIST_STATUS.OPENING;
		ELSE
			SFCReset:=FALSE;
			pistStatus:=E_PIST_STATUS.CLOSING;
		END_IF
	END_IF
	
	E_PIST_STATUS.ERROR:
	IF bInit THEN
		pistStatus:=E_PIST_STATUS.INIT;
	END_IF

		
END_CASE

ACTION _aCHECK_active_1:
IF bDepened_open1 AND bDepened_open2 THEN
	bStepDone:=TRUE;
ELSE
	bError_Condition_open:=TRUE;
	pistStatus:=E_PIST_STATUS.ERROR;
	bERROR:=TRUE;
END_IF
END_ACTION

ACTION _aCHECK_active_1_1:
IF bDepened_close1 AND bDepened_close2 THEN
	bStepDone:=TRUE;
ELSE
	pistStatus:=E_PIST_STATUS.ERROR;
	bError_Condition_close:=FALSE;
	bERROR:=TRUE;
END_IF
END_ACTION

ACTION _aCHECK_entry:
bStepDone:=FALSE;
bERROR:=FALSE;
bError_Condition_open:=FALSE;
END_ACTION

ACTION _aCHECK_entry_1:
bStepDone:=FALSE;
bERROR:=FALSE;
bError_Condition_close:=FALSE;
END_ACTION

ACTION _aCLOSE_active:
IF eType=E_PIST_TYPE.NO_SENSORS OR eType=E_PIST_TYPE.ONLY_OPEN THEN
	IF CLOSE.t>close_time THEN
		bStepDone:=TRUE;
	END_IF
END_IF

	
IF eType=E_PIST_TYPE.BOTH OR eType=E_PIST_TYPE.ONLY_CLOSE THEN	
	IF bSEN_CLOSE THEN
		bStepDone:=TRUE;
	END_IF
	IF CLOSE.t>close_timeout THEN
		bERROR:=TRUE;
		bStepDone:=TRUE;
	END_IF
END_IF
END_ACTION

ACTION _aCLOSE_entry:
bStepDone:=FALSE;
bVALVE_CLOSE:=TRUE;
bVALVE_OPEN:=FALSE;
END_ACTION

ACTION _aCLOSE_exit:
IF NOT bERROR THEN
	pistStatus:=E_PIST_STATUS.CLOSED;
ELSE
	pistStatus:=E_PIST_STATUS.ERROR;
END_IF
END_ACTION

ACTION _aNEUTRAL_entry:
pistStatus:=E_PIST_STATUS.NEUTRAL;
bVALVE_CLOSE:=FALSE;
bVALVE_OPEN:=FALSE;
END_ACTION

ACTION _aOPEN_active:
IF eType=E_PIST_TYPE.NO_SENSORS OR eType=E_PIST_TYPE.ONLY_CLOSE THEN
	IF OPEN.t>open_time THEN
		bStepDone:=TRUE;
	END_IF
END_IF

	
IF eType=E_PIST_TYPE.BOTH OR eType=E_PIST_TYPE.ONLY_OPEN THEN	
	IF bSEN_OPEN THEN
		bStepDone:=TRUE;
	END_IF
	IF OPEN.t>open_timeout THEN
		bERROR:=TRUE;
		bStepDone:=TRUE;
	END_IF
END_IF
END_ACTION

ACTION _aOPEN_entry:
bStepDone:=FALSE;
bVALVE_OPEN:=TRUE;
bVALVE_CLOSE:=FALSE;
END_ACTION

ACTION _aOPEN_exit:
IF NOT bERROR THEN
	pistStatus:=E_PIST_STATUS.OPENED;
ELSE
	pistStatus:=E_PIST_STATUS.ERROR;
END_IF
END_ACTION

ACTION _aUNNEUTRAL_entry:
bNeutral:=FALSE;
END_ACTION

ACTION A_CLOSE:
bCMD_OPEN_SWR:=FALSE;
bNeutral:=FALSE;
END_ACTION

ACTION A_INIT:
bInit:=TRUE;
bNeutral:=FALSE;
bCMD_OPEN:=bDefaultState;
bCMD_OPEN_SWR:=bDefaultState;
END_ACTION

ACTION A_NEUTRAL:
bNeutral:=TRUE;
END_ACTION

ACTION A_OPEN:
bCMD_OPEN_SWR:=TRUE;
bNeutral:=FALSE;
END_ACTION

ACTION A_UNNEUTRAL:
bNeutral:=FALSE;
END_ACTION

ACTION close_pist:
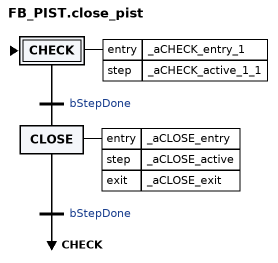
INITIAL_STEP CHECK:  // min time T#1s
    _aCHECK_entry_1(P1);  // entry action
    _aCHECK_active_1_1(N);  // step action
END_STEP
TRANSITION FROM CHECK TO CLOSE
    := bStepDone;
END_TRANSITION
STEP CLOSE:
    _aCLOSE_entry(P1);  // entry action
    _aCLOSE_active(N);  // step action
    _aCLOSE_exit(P0);  // exit action
END_STEP
TRANSITION FROM CLOSE TO CHECK
    := bStepDone;
END_TRANSITION
END_ACTION

ACTION open_pist:
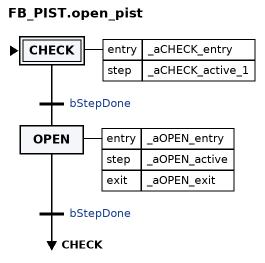
INITIAL_STEP CHECK:  // min time T#1s
    _aCHECK_entry(P1);  // entry action
    _aCHECK_active_1(N);  // step action
END_STEP
TRANSITION FROM CHECK TO OPEN
    := bStepDone;
END_TRANSITION
STEP OPEN:
    _aOPEN_entry(P1);  // entry action
    _aOPEN_active(N);  // step action
    _aOPEN_exit(P0);  // exit action
END_STEP
TRANSITION FROM OPEN TO CHECK
    := bStepDone;
END_TRANSITION
END_ACTION

END_FUNCTION_BLOCK

// ---- STATIONS/_SEPARATE.TcPOU
FUNCTION_BLOCK _SEPARATE EXTENDS FB_STATION
VAR_INPUT
	b_BULL_SENSOR:BOOL:=FALSE;
	piston_updown: REFERENCE TO FB_PIST;
	piston_colet1: REFERENCE TO FB_PIST;
	piston_colet2: REFERENCE TO FB_PIST;
	piston_colet3: REFERENCE TO FB_PIST;
	piston_colet4: REFERENCE TO FB_PIST;
	piston_puller: REFERENCE TO FB_PIST;
	piston_tray: REFERENCE TO FB_PIST;
	piston_pins: REFERENCE TO FB_PIST;
	piston_tray_door: REFERENCE TO FB_PIST;
	piston_tray_push: REFERENCE TO FB_PIST;
	bInit:BOOL:=FALSE;
	
	
	fbAxis:REFERENCE TO FB_Axis;
	
END_VAR
VAR_OUTPUT
	bRUNNING:BOOL :=FALSE;
	bError:BOOL:=FALSE;
END_VAR
VAR
	//bHomed:BOOL :=FALSE;
	tDelay: TON;
	bDELAY: BOOL:=FALSE;
	E: INT;
	
	//bDone: BOOL;
	step_timeout: TIME:=T#7S;
	colet_close: INT;
END_VAR


act();

CASE eState OF
	
	E_STATION_STATE.homing:
		//SFCReset:=FALSE;
		//SFCInit:=FALSE;
		piston_updown.A_INIT();
		piston_colet1.A_INIT(); piston_colet2.A_INIT();piston_colet3.A_INIT();piston_colet4.A_INIT();
		piston_tray.A_INIT();
		piston_tray_push.A_INIT();
		piston_tray_door.A_INIT();
		piston_pins.A_INIT();
		eState:= E_STATION_STATE.idle;
		bHomed:=TRUE;
		bError:=FALSE;
		//axis-------------------
		fbAxis.bEnable:=TRUE;
		fbAxis.bHalt:=FALSE;
		fbAxis.bSetPosition:=FALSE;
		fbAxis.bReset:=FALSE;
		
	E_STATION_STATE.uninit:
		eState:= E_STATION_STATE.homing;
		fbAxis.bDo_Step_FW:=FALSE;
		fbAxis.bMoveRel:=FALSE;
		fbAxis.stepFW_state:=0;
		fbAxis.bHalt:=FALSE;
		fbAxis.bReset:=FALSE;

	E_STATION_STATE.idle:
		//idle
		
	E_STATION_STATE.do_action1://delay and lower device
		//main action
		
	E_STATION_STATE.done:
		//dd
	 
	E_STATION_STATE.pause:
		//paused
	
	E_STATION_STATE.error:
		//error
	
	E_STATION_STATE.estop:
		fbAxis.stepFW_state:=0;
		fbAxis.bHalt:=TRUE;
		fbAxis.bReset:=TRUE;
		bHomed:=FALSE;

END_CASE

ACTION _aCLOSE_COLET_1_4_active:
IF  NOT (eState = E_STATION_STATE.pause) THEN
bDone:=TRUE;
END_IF
END_ACTION

ACTION _aCLOSE_COLET_1_4_entry:

	bDone:=FALSE;
	IF NOT (eState = E_STATION_STATE.pause) THEN
		piston_colet1.A_OPEN();
		piston_colet4.A_OPEN();
		piston_pins.A_OPEN();
		
	END_IF
END_ACTION

ACTION _aCLOSE_COLET_active:
IF NOT (eState = E_STATION_STATE.pause) THEN

//IF piston_colet1.pistStatus= E_PIST_STATUS.OPENED AND piston_colet2.pistStatus= E_PIST_STATUS.OPENED THEN
	bDone:=TRUE;
//END_IF

END_IF
END_ACTION

ACTION _aCLOSE_COLET_entry:

	bDone:=FALSE;
	IF NOT (eState = E_STATION_STATE.pause) THEN
		piston_colet2.A_OPEN();
		piston_colet3.A_OPEN();
		
	END_IF
END_ACTION

ACTION _aIDLE_active:
IF eState = E_STATION_STATE.do_action1 THEN 
	bDone:=TRUE;
	
END_IF
END_ACTION

ACTION _aIDLE_entry:
bDone:=FALSE;
END_ACTION

ACTION _aJACK_UP1_active:
IF JACK_UP1.t>step_timeout AND NOT (eState = E_STATION_STATE.pause)THEN
		bERROR:=TRUE;
END_IF
IF fbAxis.RELATIVE.Done THEN
	bDone:=TRUE;
END_IF
END_ACTION

ACTION _aJACK_UP1_entry:

	bDone:=FALSE;
	IF NOT (eState = E_STATION_STATE.pause) THEN
		piston_updown.A_NEUTRAL();
		fbAxis.bDo_Step_FW:=TRUE;
		
	END_IF
END_ACTION

ACTION _aJACK_UP2_active:
IF JACK_UP2.t>step_timeout AND NOT (eState = E_STATION_STATE.pause) THEN
		bERROR:=TRUE;
END_IF
IF fbAxis.RELATIVE.Done THEN
	bDone:=TRUE;
END_IF
END_ACTION

ACTION _aJACK_UP2_entry:

	bDone:=FALSE;
	IF NOT (eState = E_STATION_STATE.pause) THEN
		fbAxis.bDo_Step_FW:=TRUE;
		
	END_IF
END_ACTION

ACTION _aLOWER_LIFT_active:
IF LOWER_LIFT.t>step_timeout AND NOT (eState = E_STATION_STATE.pause) THEN
		bERROR:=TRUE;
END_IF

IF piston_updown.pistStatus= E_PIST_STATUS.OPENED   THEN
	bDone:=TRUE;
END_IF
END_ACTION

ACTION _aLOWER_LIFT_entry:

	bDone:=FALSE;
	IF NOT bSkip AND NOT (eState = E_STATION_STATE.pause) THEN
		piston_updown.A_OPEN();	
		
	ELSE
		eState:=E_STATION_STATE.done;
	END_IF
END_ACTION

ACTION _aOPEN_COLETS_active:
IF OPEN_COLETS.t>step_timeout AND NOT (eState = E_STATION_STATE.pause) THEN
		bERROR:=TRUE;
END_IF

IF piston_colet1.pistStatus= E_PIST_STATUS.CLOSED AND piston_colet2.pistStatus= E_PIST_STATUS.CLOSED AND piston_colet3.pistStatus= E_PIST_STATUS.CLOSED AND piston_colet4.pistStatus= E_PIST_STATUS.CLOSED THEN
	bDone:=TRUE;
END_IF
END_ACTION

ACTION _aOPEN_COLETS_entry:

	bDone:=FALSE;
	IF NOT (eState = E_STATION_STATE.pause) THEN
		piston_colet2.A_CLOSE();
		piston_colet3.A_CLOSE();
		piston_colet1.A_CLOSE();
		piston_colet4.A_CLOSE();
		
	END_IF
END_ACTION

ACTION _aPINS_DOWN_active:
IF PINS_DOWN.t>step_timeout AND NOT (eState = E_STATION_STATE.pause) THEN
		bERROR:=TRUE;
END_IF

IF piston_pins.pistStatus= E_PIST_STATUS.OPENED THEN
	bDone:=TRUE;
END_IF
END_ACTION

ACTION _aPINS_DOWN_entry:

	bDone:=FALSE;
	IF NOT (eState = E_STATION_STATE.pause) THEN
		piston_pins.A_OPEN();
	END_IF
END_ACTION

ACTION _aPINS_UP_active:
IF PINS_UP.t>step_timeout AND NOT (eState = E_STATION_STATE.pause) THEN
		bERROR:=TRUE;
END_IF

IF piston_pins.pistStatus= E_PIST_STATUS.CLOSED THEN
	bDone:=TRUE;
END_IF
END_ACTION

ACTION _aPINS_UP_entry:

	bDone:=FALSE;
	IF NOT (eState = E_STATION_STATE.pause) THEN
		piston_pins.A_CLOSE();
	END_IF
END_ACTION

ACTION _aRAISE_LIFT_active:
IF RAISE_LIFT.t>step_timeout AND NOT (eState = E_STATION_STATE.pause) THEN
		bERROR:=TRUE;
END_IF

IF piston_updown.pistStatus= E_PIST_STATUS.CLOSED THEN
	bDone:=TRUE;
END_IF
END_ACTION

ACTION _aRAISE_LIFT_entry:

	bDone:=FALSE;
	IF NOT (eState = E_STATION_STATE.pause) THEN
		piston_updown.A_CLOSE();
	END_IF
END_ACTION

ACTION _aTRAY_active:
IF TRAY.t>step_timeout AND NOT (eState = E_STATION_STATE.pause) THEN
		bERROR:=TRUE;
END_IF

IF piston_tray.pistStatus= E_PIST_STATUS.OPENED THEN
	bDone:=TRUE;
END_IF
END_ACTION

ACTION _aTRAY_entry:

	bDone:=FALSE;
	IF NOT (eState = E_STATION_STATE.pause) THEN
		piston_tray.A_OPEN();
	END_IF
END_ACTION

ACTION _aTRAY_JACK_BACK_active:
IF NOT (eState = E_STATION_STATE.pause) THEN
	eState:= E_STATION_STATE.done;
	bDone:=TRUE;
END_IF
END_ACTION

ACTION _aUNINIT_entry:
bDone:=TRUE;
END_ACTION

ACTION act:
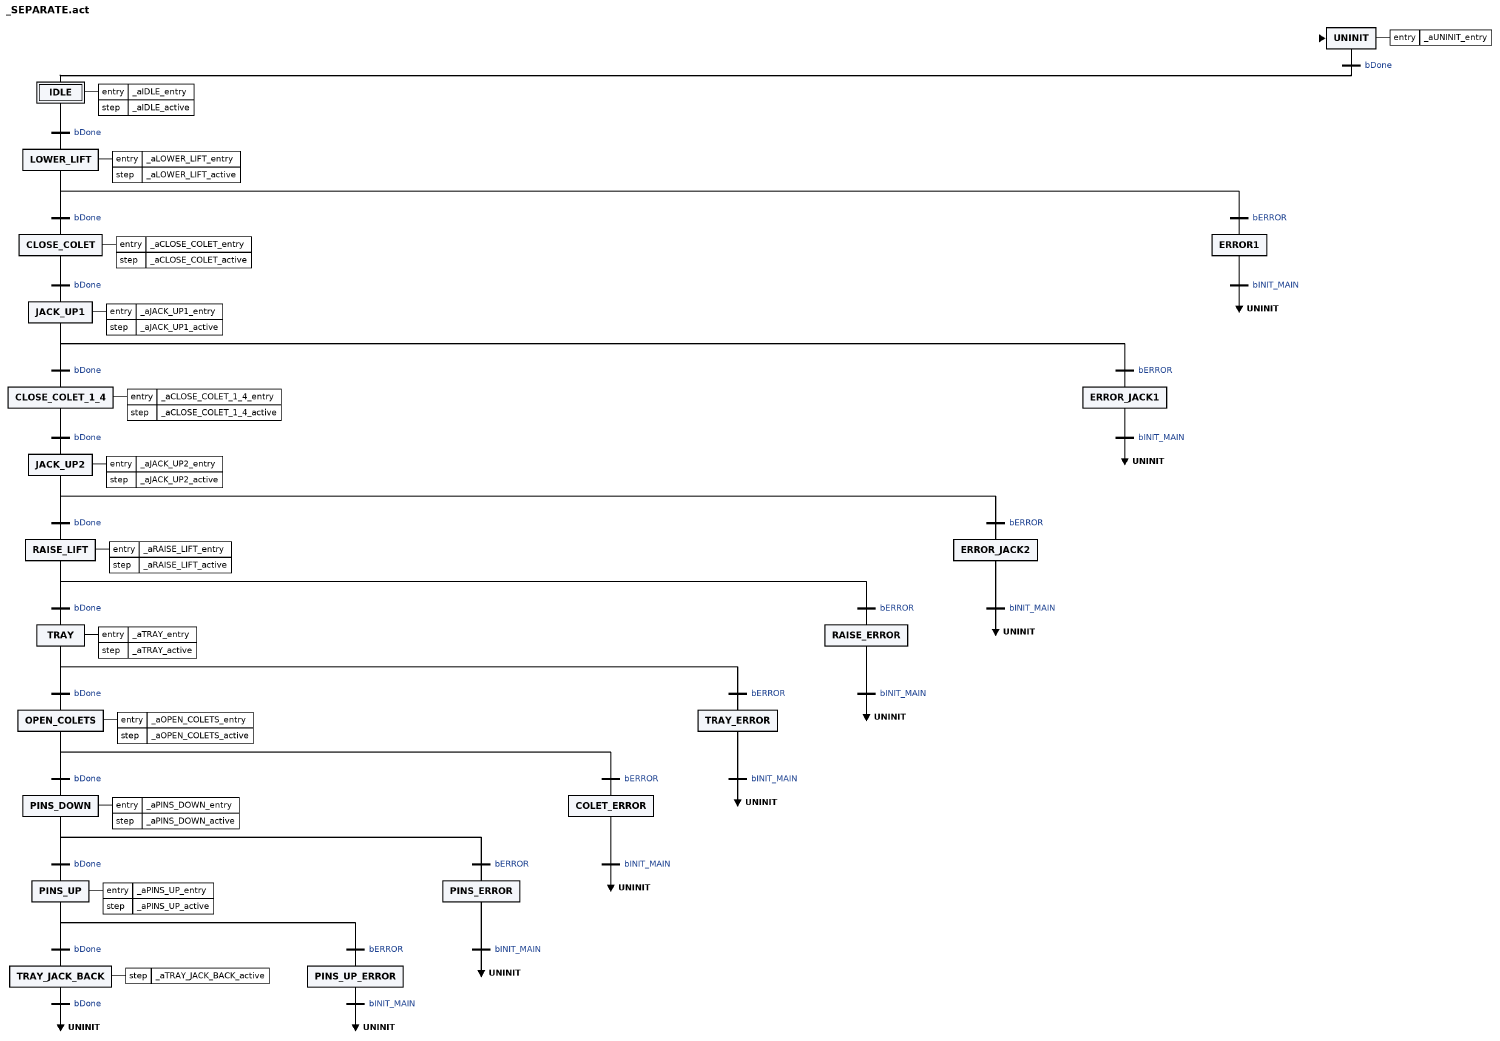
STEP UNINIT:
    _aUNINIT_entry(P1);  // entry action
END_STEP
TRANSITION FROM UNINIT TO IDLE
    := bDone;
END_TRANSITION
INITIAL_STEP IDLE:
    _aIDLE_entry(P1);  // entry action
    _aIDLE_active(N);  // step action
END_STEP
TRANSITION FROM IDLE TO LOWER_LIFT
    := bDone;
END_TRANSITION
STEP LOWER_LIFT:
    _aLOWER_LIFT_entry(P1);  // entry action
    _aLOWER_LIFT_active(N);  // step action
END_STEP
TRANSITION FROM LOWER_LIFT TO CLOSE_COLET
    := bDone;
END_TRANSITION
STEP CLOSE_COLET:  // min time T#1s
    _aCLOSE_COLET_entry(P1);  // entry action
    _aCLOSE_COLET_active(N);  // step action
END_STEP
TRANSITION FROM CLOSE_COLET TO JACK_UP1
    := bDone;
END_TRANSITION
STEP JACK_UP1:  // min time T#2s
    _aJACK_UP1_entry(P1);  // entry action
    _aJACK_UP1_active(N);  // step action
END_STEP
TRANSITION FROM JACK_UP1 TO CLOSE_COLET_1_4
    := bDone;
END_TRANSITION
STEP CLOSE_COLET_1_4:
    _aCLOSE_COLET_1_4_entry(P1);  // entry action
    _aCLOSE_COLET_1_4_active(N);  // step action
END_STEP
TRANSITION FROM CLOSE_COLET_1_4 TO JACK_UP2
    := bDone;
END_TRANSITION
STEP JACK_UP2:  // min time T#2s
    _aJACK_UP2_entry(P1);  // entry action
    _aJACK_UP2_active(N);  // step action
END_STEP
TRANSITION FROM JACK_UP2 TO RAISE_LIFT
    := bDone;
END_TRANSITION
STEP RAISE_LIFT:
    _aRAISE_LIFT_entry(P1);  // entry action
    _aRAISE_LIFT_active(N);  // step action
END_STEP
TRANSITION FROM RAISE_LIFT TO TRAY
    := bDone;
END_TRANSITION
STEP TRAY:
    _aTRAY_entry(P1);  // entry action
    _aTRAY_active(N);  // step action
END_STEP
TRANSITION FROM TRAY TO OPEN_COLETS
    := bDone;
END_TRANSITION
STEP OPEN_COLETS:
    _aOPEN_COLETS_entry(P1);  // entry action
    _aOPEN_COLETS_active(N);  // step action
END_STEP
TRANSITION FROM OPEN_COLETS TO PINS_DOWN
    := bDone;
END_TRANSITION
TRANSITION FROM OPEN_COLETS TO COLET_ERROR
    := bERROR;
END_TRANSITION
STEP COLET_ERROR:
END_STEP
TRANSITION FROM COLET_ERROR TO UNINIT
    := bINIT_MAIN;
END_TRANSITION
STEP PINS_DOWN:
    _aPINS_DOWN_entry(P1);  // entry action
    _aPINS_DOWN_active(N);  // step action
END_STEP
TRANSITION FROM PINS_DOWN TO PINS_UP
    := bDone;
END_TRANSITION
STEP PINS_UP:
    _aPINS_UP_entry(P1);  // entry action
    _aPINS_UP_active(N);  // step action
END_STEP
TRANSITION FROM PINS_UP TO TRAY_JACK_BACK
    := bDone;
END_TRANSITION
STEP TRAY_JACK_BACK:
    _aTRAY_JACK_BACK_active(N);  // step action
END_STEP
TRANSITION FROM TRAY_JACK_BACK TO UNINIT
    := bDone;
END_TRANSITION
TRANSITION FROM PINS_UP TO PINS_UP_ERROR
    := bERROR;
END_TRANSITION
STEP PINS_UP_ERROR:
END_STEP
TRANSITION FROM PINS_UP_ERROR TO UNINIT
    := bINIT_MAIN;
END_TRANSITION
TRANSITION FROM PINS_DOWN TO PINS_ERROR
    := bERROR;
END_TRANSITION
STEP PINS_ERROR:
END_STEP
TRANSITION FROM PINS_ERROR TO UNINIT
    := bINIT_MAIN;
END_TRANSITION
TRANSITION FROM TRAY TO TRAY_ERROR
    := bERROR;
END_TRANSITION
STEP TRAY_ERROR:
END_STEP
TRANSITION FROM TRAY_ERROR TO UNINIT
    := bINIT_MAIN;
END_TRANSITION
TRANSITION FROM RAISE_LIFT TO RAISE_ERROR
    := bERROR;
END_TRANSITION
STEP RAISE_ERROR:
END_STEP
TRANSITION FROM RAISE_ERROR TO UNINIT
    := bINIT_MAIN;
END_TRANSITION
TRANSITION FROM JACK_UP2 TO ERROR_JACK2
    := bERROR;
END_TRANSITION
STEP ERROR_JACK2:
END_STEP
TRANSITION FROM ERROR_JACK2 TO UNINIT
    := bINIT_MAIN;
END_TRANSITION
TRANSITION FROM JACK_UP1 TO ERROR_JACK1
    := bERROR;
END_TRANSITION
STEP ERROR_JACK1:
END_STEP
TRANSITION FROM ERROR_JACK1 TO UNINIT
    := bINIT_MAIN;
END_TRANSITION
TRANSITION FROM LOWER_LIFT TO ERROR1
    := bERROR;
END_TRANSITION
STEP ERROR1:
END_STEP
TRANSITION FROM ERROR1 TO UNINIT
    := bINIT_MAIN;
END_TRANSITION
// branch label Branch7_act
// branch label Branch8_act
// branch label Branch6_act
// branch label Branch5_act
// branch label Branch4_act
// branch label Branch3_act
// branch label Branch2_act
// branch label Branch0_act
END_ACTION

END_FUNCTION_BLOCK

// ---- POUs/AXES/FB_Axis.TcPOU
FUNCTION_BLOCK FB_Axis
VAR_INPUT
	sName:STRING;
	Axis:Axis_ref;
	bEnable:BOOL:=FALSE;
	bHalt:BOOL:=FALSE;
	bHome:BOOL:=FALSE;
	bReset:BOOL:=FALSE;
	bSetPosition:BOOL:=FALSE;
	Dist:REAL;
	bMoveRel:BOOL:=FALSE;
	bMoveRelBusy:BOOL;
	rPos:LREAL;
	rVel:LREAL;
	rAcc:LREAL;
	rDec:LREAL;
	jJerk:LREAL;
	bMoveABS:BOOL:=FALSE;
	bMoveAbsBusy:BOOL;
	bJogPos:BOOL;
	bJogNeg:BOOL;
	rStep: REAL:=400;
	rStep_vel: REAL:=400;
	bmanual:BOOL:=FALSE;
	bDo_Step_FW:BOOL:=FALSE;
	bDo_Step_BW:BOOL:=FALSE;
	stepFW_state:INT:=0;
	stepBW_state:INT:=0;
	bStop:BOOL:=0;
	bHomeBusy:BOOL;
	ton_Reset: TON;
END_VAR

VAR_OUTPUT
	bBusy: BOOL;
	bError:BOOL;
	bInPos:BOOL;
	rActPos:LREAL;
	rActVel:LREAL;
	bRelDone:BOOL;
	bAbsDone:BOOL;
END_VAR
VAR
	tDelay: TON;
	bDelay:BOOL:=FALSE;
	MoveAbsolute: MC_MoveAbsolute;
	power: MC_Power;
	Reset: MC_Reset;
	SetPosition: MC_SetPosition;
	JOG: MC_Jog;
	RELATIVE: MC_MoveRelative;
	HALT: MC_Halt;
	HOME: MC_Home;
	bFirst_run:BOOL:=FALSE;
	bStopBusy:BOOL;
	
	
	
	
END_VAR

IF NOT bFirst_run THEN
	RESET.Execute:=TRUE;
END_IF


rActPos:=Axis.NcToPlc.ActPos;
rActVel:=Axis.NcToPlc.ActVelo;

STEP_FW();


IF RELATIVE.Busy OR JOG.Busy OR moveAbsolute.busy THEN
	bBusy:=TRUE;
ELSE
	bBusy:=FALSE;
END_IF

IF POWER.error OR RELATIVE.error OR MoveAbsolute.error OR JOG.error THEN
	bError:=TRUE;
ELSE
	bError:=FALSE;
END_IF

IF RELATIVE.Done OR JOG.Done OR moveAbsolute.Done THEN
	bInPos:=TRUE;
ELSE
	bInPos:=FALSE;
END_IF
motion_commands();
(*
RELATIVE(
	Axis:= Axis, 
	Execute:=bMoveRel , 
	Distance:= Dist, 
	Velocity:=rVel , 
	Acceleration:= , 
	Deceleration:= , 
	Jerk:= , 
	BufferMode:= , 
	Options:= , 
	Done=> bRelDone, 
	Busy=> , 
	Active=> , 
	CommandAborted=> , 
	Error=> , 
	ErrorID=> );
	
JOG(
	Axis:=Axis , 
	JogForward:= bJogPos, 
	JogBackwards:=bJogNeg , 
	Mode:= E_JogMode.MC_JOGMODE_CONTINOUS,
	Position:=rPos , 
	Velocity:= rVel, 
	Acceleration:= , 
	Deceleration:= , 
	Jerk:= , 
	Done=> , 
	Busy=> , 
	Active=> , 
	CommandAborted=> , 
	Error=> , 
	ErrorID=> );

Power(
	Axis:= Axis, 
	Enable:= bEnable, 
	Enable_Positive:= bEnable, 
	Enable_Negative:= bEnable, 
	Override:= 100, 
	BufferMode:= , 
	Options:= , 
	Status=> , 
	Busy=> , 
	Active=> , 
	Error=> , 
	ErrorID=> );

Reset(
	Axis:= Axis, 
	Execute:= bReset, 
	Done=> , 
	Busy=> , 
	Error=> , 
	ErrorID=> );
	
SetPosition(
	Axis:= Axis, 
	Execute:= bSetPosition, 
	Position:= rPos, 
	Mode:= , 
	Options:= , 
	Done=> , 
	Busy=> , 
	Error=> , 
	ErrorID=> );

MoveAbsolute(
	Axis:= Axis, 
	Execute:= bMoveABS, 
	Position:= rPos, 
	Velocity:= rVel, 
	Acceleration:= , 
	Deceleration:= , 
	Jerk:= , 
	BufferMode:= , 
	Options:= , 
	Done=> bAbsDone, 
	Busy=> , 
	Active=> , 
	CommandAborted=> , 
	Error=> , 
	ErrorID=> );
	
HALT(
	Axis:= Axis, 
	Execute:= bHalt, 
	Deceleration:= , 
	Jerk:= , 
	BufferMode:= , 
	Options:= , 
	Done=> , 
	Busy=> , 
	Active=> , 
	CommandAborted=> , 
	Error=> , 
	ErrorID=> );

	*)

METHOD clear_cmd_req : BOOL
VAR_INPUT
END_VAR

bMoveABS:= bMoveRel:= bJogPos:= bJogNeg:=FALSE;
END_METHOD

ACTION motion_commands:
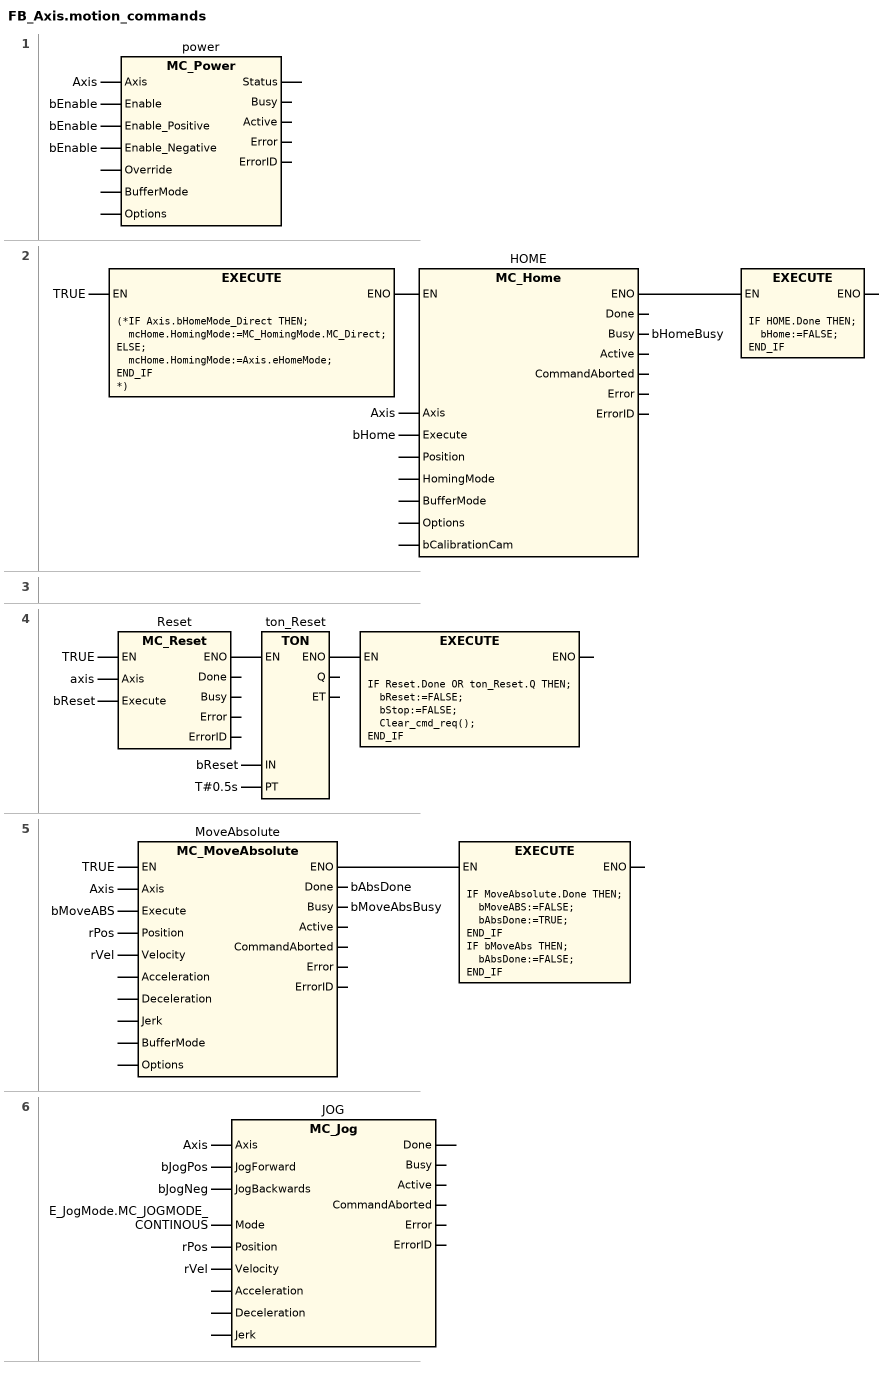
// NETWORK 1
power(Axis := Axis, Enable := bEnable, Enable_Positive := bEnable, Enable_Negative := bEnable); // MC_Power

// NETWORK 2

(*IF Axis.bHomeMode_Direct THEN;
	mcHome.HomingMode:=MC_HomingMode.MC_Direct;
ELSE;
	mcHome.HomingMode:=Axis.eHomeMode;
END_IF
*)
HOME(Axis := Axis, Execute := bHome, Busy => bHomeBusy); // MC_Home

IF HOME.Done THEN;
	bHome:=FALSE;
END_IF

// NETWORK 3

// NETWORK 4
Reset(Axis := axis, Execute := bReset); // MC_Reset
ton_Reset(IN := bReset, PT := T#0.5s); // TON

IF Reset.Done OR ton_Reset.Q THEN;
	bReset:=FALSE;
	bStop:=FALSE;
	Clear_cmd_req();
END_IF

// NETWORK 5
MoveAbsolute(
    Axis := Axis,
    Execute := bMoveABS,
    Position := rPos,
    Velocity := rVel,
    Done => bAbsDone,
    Busy => bMoveAbsBusy); // MC_MoveAbsolute

IF MoveAbsolute.Done THEN;
	bMoveABS:=FALSE;
	bAbsDone:=TRUE;
END_IF
IF bMoveAbs THEN;
	bAbsDone:=FALSE;
END_IF

// NETWORK 6
JOG(
    Axis := Axis,
    JogForward := bJogPos,
    JogBackwards := bJogNeg,
    Mode := E_JogMode.MC_JOGMODE_CONTINOUS,
    Position := rPos,
    Velocity := rVel); // MC_Jog

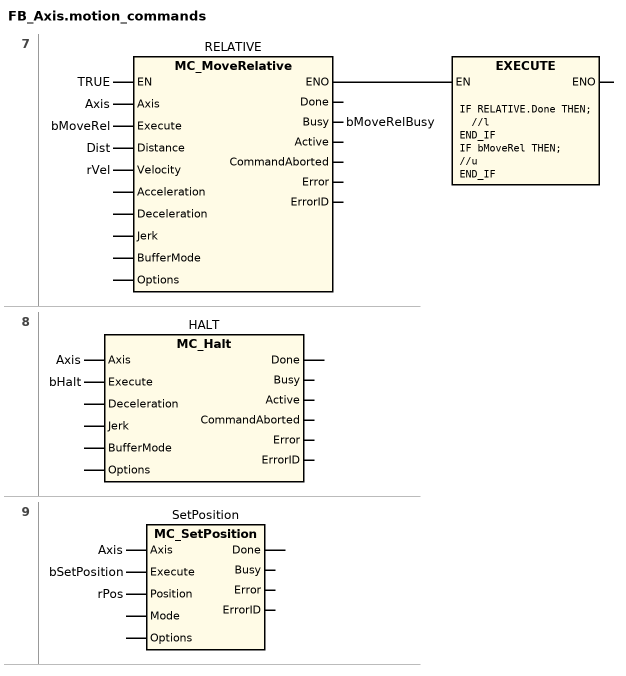
// NETWORK 7
RELATIVE(Axis := Axis, Execute := bMoveRel, Distance := Dist, Velocity := rVel, Busy => bMoveRelBusy); // MC_MoveRelative

IF RELATIVE.Done THEN;
	//l
END_IF
IF bMoveRel THEN;
//u
END_IF

// NETWORK 8
HALT(Axis := Axis, Execute := bHalt); // MC_Halt

// NETWORK 9
SetPosition(Axis := Axis, Execute := bSetPosition, Position := rPos); // MC_SetPosition
END_ACTION

METHOD STEP_FW : BOOL
VAR_INPUT
END_VAR
  
CASE stepFW_state OF
	
	0:
	IF bDo_Step_FW AND NOT bManual THEN		
		bMoveRel:=FALSE;
		//bReset:=TRUE;
		bDo_Step_FW:=FALSE;
		stepFW_state := 1;	
	END_IF

	1:
	Dist:=rStep;
	rVel:=rStep_Vel;
	bEnable:=TRUE;
	bMoveRel:=FALSE;
	stepFW_state := 2;
	//bReset:=FALSE;
	
	2:
	bMoveRel:=TRUE;
	stepFW_state := 3;
	
	3:
	IF RELATIVE.Done THEN
		 bDo_Step_FW:=FALSE;
		 stepFW_state := 0;
	END_IF
	
	
	
	
END_CASE
END_METHOD

END_FUNCTION_BLOCK

// ---- STATIONS/FB_CLEAN.TcPOU
FUNCTION_BLOCK FB_CLEAN EXTENDS FB_STATION
VAR_INPUT
	pClean: REFERENCE TO FB_PIST;
END_VAR
VAR_OUTPUT
END_VAR
VAR
END_VAR


CASE eCLEAN OF
	E_STATION_STATE.homing:
		pClean.A_INIT();
		bHomed:=TRUE;
		eCLEAN:= E_STATION_STATE.idle;
		
	E_STATION_STATE.uninit:
		eCLEAN:= E_STATION_STATE.idle;

	E_STATION_STATE.idle:
		//fdgdfgfdgf
			
	E_STATION_STATE.do_action1:
		IF NOT bSkip THEN
			pClean.A_OPEN();
			eCLEAN:=E_STATION_STATE.do_action2;
		ELSE
			eCLEAN:=E_STATION_STATE.done;
		END_IF
		
		
	E_STATION_STATE.do_action2:
		IF pClean.PistStatus= E_PIST_STATUS.OPENED THEN
			eCLEAN:=E_STATION_STATE.do_action3;
		END_IF
		
	E_STATION_STATE.do_action3:
		pClean.A_CLOSE();
		eCLEAN:=E_STATION_STATE.do_action4;
		
	E_STATION_STATE.do_action4:
		IF pClean.PistStatus= E_PIST_STATUS.CLOSED  THEN
			eCLEAN:=E_STATION_STATE.done;
		END_IF
	
	
	E_STATION_STATE.done:
		//done
		
	E_STATION_STATE.pause:
		//paused

END_CASE

END_FUNCTION_BLOCK

// ---- STATIONS/FB_DROP.TcPOU
FUNCTION_BLOCK FB_DROP EXTENDS FB_STATION
VAR_INPUT
	pPush: REFERENCE TO FB_PIST;
	pOpen1: REFERENCE TO FB_PIST;
	pOpen2: REFERENCE TO FB_PIST;
END_VAR
VAR_OUTPUT
END_VAR
VAR
END_VAR

CASE eDROP OF
	E_STATION_STATE.homing:
		pOpen1.A_INIT();
		pOpen2.A_INIT();
		pPush.A_INIT();
		bHomed:=TRUE;
		eDROP:= E_STATION_STATE.idle;
		
	E_STATION_STATE.uninit:
		eDROP:= E_STATION_STATE.idle;

	E_STATION_STATE.idle:
		//fdgdfgfdgf
			
	E_STATION_STATE.do_action1:
		IF NOT bSkip THEN
			pOpen1.A_OPEN();
			pOpen2.A_OPEN();
			eDROP:=E_STATION_STATE.do_action2;
		ELSE
			eDROP:=E_STATION_STATE.done;
		END_IF
		
		
	E_STATION_STATE.do_action2:
		IF pOpen1.PistStatus= E_PIST_STATUS.OPENED AND pOpen2.PistStatus= E_PIST_STATUS.OPENED THEN
			pPush.A_OPEN();
			eDROP:=E_STATION_STATE.do_action3;
		END_IF
	
	E_STATION_STATE.do_action3:
		IF pPush.PistStatus= E_PIST_STATUS.OPENED THEN
			eDROP:=E_STATION_STATE.do_action4;
			pOpen1.A_CLOSE();
			pOpen2.A_CLOSE();
		END_IF
	
	E_STATION_STATE.do_action4:
		IF pOpen1.PistStatus= E_PIST_STATUS.CLOSED AND pOpen2.PistStatus= E_PIST_STATUS.CLOSED THEN
			pPush.A_CLOSE();
			eDROP:=E_STATION_STATE.do_action5;
		END_IF

	E_STATION_STATE.do_action5:
		IF pPush.PistStatus= E_PIST_STATUS.CLOSED THEN
			eDROP:=E_STATION_STATE.done;
		END_IF
		
	E_STATION_STATE.done:
		//done
		
	E_STATION_STATE.pause:
		//paused

END_CASE

END_FUNCTION_BLOCK

// ---- STATIONS/FB_SUPPLY.TcPOU
FUNCTION_BLOCK FB_SUPPLY EXTENDS FB_STATION
VAR_INPUT
	
	pPush: REFERENCE TO FB_PIST;
	pLock1:REFERENCE TO FB_PIST;
	pLock2:REFERENCE TO FB_PIST;
	pOpen1:REFERENCE TO FB_PIST;
	pOpen2:REFERENCE TO FB_PIST;
	
END_VAR
VAR_OUTPUT
END_VAR
VAR
END_VAR

CASE eSUPPLY OF
	E_STATION_STATE.homing:
		pPush.A_INIT(); pLock1.A_INIT(); pLock2.A_INIT(); pOpen1.A_INIT(); pOpen2.A_INIT();
		bHomed:=TRUE;
		eSUPPLY:= E_STATION_STATE.idle;
		
	E_STATION_STATE.uninit:
		eSUPPLY:= E_STATION_STATE.homing;

	E_STATION_STATE.idle:
		//
			
	E_STATION_STATE.do_action1:
		IF NOT bSkip THEN
			
			pLock1.A_OPEN();
			pLock2.A_OPEN();
			eSUPPLY:=E_STATION_STATE.do_action2;
		ELSE
			eSUPPLY:=E_STATION_STATE.done;
		END_IF
		
	E_STATION_STATE.do_action2:	
		IF pLock1.PistStatus= E_PIST_STATUS.OPENED  AND  pLock2.PistStatus= E_PIST_STATUS.OPENED THEN
			pOpen1.A_OPEN();	
			pOpen2.A_OPEN();		
			eSUPPLY:=E_STATION_STATE.do_action3;
		END_IF
	
	E_STATION_STATE.do_action3:	
		IF pOpen1.PistStatus= E_PIST_STATUS.OPENED AND  pOpen2.PistStatus= E_PIST_STATUS.OPENED THEN
			pPush.A_OPEN();			
			eSUPPLY:=E_STATION_STATE.do_action4;
		END_IF
	
	E_STATION_STATE.do_action4:	
		IF pPush.PistStatus= E_PIST_STATUS.OPENED  THEN
			pOpen1.A_CLOSE();	
			pOpen2.A_CLOSE();	
			pLock1.A_CLOSE();
			pLock2.A_CLOSE();
			pPush.A_CLOSE();		
			eSUPPLY:=E_STATION_STATE.do_action5;
		END_IF
		
	E_STATION_STATE.do_action5:	
		IF pLock1.PistStatus= E_PIST_STATUS.CLOSED AND pLock2.PistStatus= E_PIST_STATUS.CLOSED AND pOpen1.PistStatus= E_PIST_STATUS.CLOSED AND pOpen2.PistStatus= E_PIST_STATUS.CLOSED AND pPush.PistStatus= E_PIST_STATUS.CLOSED  THEN
			eSUPPLY:=E_STATION_STATE.done;
		END_IF
	
	
	
	
	E_STATION_STATE.done:
		//
		
	E_STATION_STATE.pause:
		//paused

END_CASE

END_FUNCTION_BLOCK

// ---- STATIONS/FB_MAIN_CONV.TcPOU
FUNCTION_BLOCK FB_MAIN_CONV EXTENDS FB_STATION
VAR_INPUT
	fbAxis:REFERENCE TO FB_Axis;
END_VAR
VAR_OUTPUT
END_VAR
VAR
	rtrig_ERROR: R_TRIG;
	rtrigFW: R_TRIG;
	bStepFW:BOOL:=FALSE;
	//bStepBW:BOOL:=FALSE;
	bMOVE:BOOL :=FALSE;
	tNext: TON;
	tDelay: TON;
	bDELAY: BOOL:=FALSE;
	counter: INT;
	counter1: INT;
	bTest: INT;
	bSTARTUP: BOOL;
	total_length: INT;
	cart_space: INT;
	inc: INT;
	state: INT;
	temp: INT;
END_VAR

FOR counter:=1 TO num_of_carts BY 1 DO
	fbCART[counter]();
END_FOR;
rtrigFW(CLK:= bStepFW, Q=> );

IF NOT bFirstRun THEN
	A_set_cart_spaces();
	A_SETUP();
	bFirstRun:=TRUE;
END_IF

IF rtrigFW.Q AND (eMAIN_CONVAYOR_STATE =E_CONVAYOR_STATE.pause OR eMAIN_CONVAYOR_STATE =E_CONVAYOR_STATE.done)  THEN
	eMAIN_CONVAYOR_STATE:=E_CONVAYOR_STATE.do_move;
END_IF


tDelay(IN:=bDELAY);
tNext(IN:=bMOVE , PT:=T#1S , Q=> , ET=> );

CASE eMAIN_CONVAYOR_STATE OF
	E_CONVAYOR_STATE.homing:
		bHomed:=TRUE;
		eMAIN_CONVAYOR_STATE:=E_CONVAYOR_STATE.idle;
		fbAxis.bEnable:=TRUE;
		fbAxis.bHalt:=FALSE;
		bDELAY:=FALSE;
		fbAxis.bSetPosition:=FALSE;
		fbAxis.bReset:=FALSE;
	
	E_CONVAYOR_STATE.uninit:
		IF NOT  bHomed THEN
			eMAIN_CONVAYOR_STATE:=E_CONVAYOR_STATE.homing;
		ELSE
			eMAIN_CONVAYOR_STATE:=E_CONVAYOR_STATE.idle;	
		END_IF
		fbAxis.bDo_Step_FW:=FALSE;
		fbAxis.bMoveRel:=FALSE;
		fbAxis.stepFW_state:=0;
		fbAxis.bHalt:=FALSE;
		fbAxis.bReset:=FALSE;
		
	E_CONVAYOR_STATE.idle:
		//
	
	E_CONVAYOR_STATE.do_move:
		eMAIN_CONVAYOR_STATE:=E_CONVAYOR_STATE.st1;
		
	
	E_CONVAYOR_STATE.st1: // start motion
		IF NOT fbAxis.bBusy  AND NOT fbAxis.bError THEN
			fbAxis.rPos:=0;	
			fbAxis.bSetPosition:=TRUE;	
			A_CARTS_STEP();
			fbAxis.bDo_Step_FW:=TRUE;
			eMAIN_CONVAYOR_STATE:=E_CONVAYOR_STATE.st2;
		END_IF
		
	E_CONVAYOR_STATE.st2:
		IF fbAxis.rActPos < 200 THEN
			eMAIN_CONVAYOR_STATE:=E_CONVAYOR_STATE.st3;	
			fbAxis.bSetPosition:=FALSE;
		END_IF
		
	E_CONVAYOR_STATE.st3:
		IF fbAxis.rActPos > (fbAxis.rStep/2)	THEN
			A_CARTS_STEP();	
			eMAIN_CONVAYOR_STATE:=E_CONVAYOR_STATE.st4;
		END_IF


	E_CONVAYOR_STATE.st4:
		IF fbAxis.bInPos THEN
			eMAIN_CONVAYOR_STATE:=E_CONVAYOR_STATE.done;
		END_IF
		
	E_CONVAYOR_STATE.done:
		//...
	
	E_CONVAYOR_STATE.pause:
	//
	
	E_CONVAYOR_STATE.estop:
		fbAxis.stepFW_state:=0;
		fbAxis.bHalt:=TRUE;
		fbAxis.bReset:=TRUE;
		bHomed:=FALSE;
	//...
	
	E_CONVAYOR_STATE.error:
		//...
		
	rtrig_ERROR(CLK:=(eMAIN_CONVAYOR_STATE=E_CONVAYOR_STATE.error), Q=> );
	IF rtrig_ERROR.Q THEN
		gEventType:= 'Alarm'; 
		gEventSeverity:= 'Error';
		gEventIdentity:=2001;
		gEventName:= 'MAIN CONVAYOR';
		gEventText:='MOTOR ERROR:';
		fbEventLogger.mAdd();
	END_IF
	
END_CASE

ACTION A_CARTS_STEP:
FOR counter1:=1 TO num_of_carts BY 1 DO
	fbCART[counter1].A_STEP();
END_FOR;
END_ACTION

ACTION A_set_cart_spaces:
 total_length := (conv_height*2)+(conv_length*2);
cart_space := total_length /((num_of_carts*2));
inc:=1;
posArrX[inc]:= 0+X_OFFSET;
posArrY[inc]:= 0+(conv_height/2)+Y_OFFSET;



WHILE state = 0 DO    //left1
	IF posArrY[inc]-cart_space < Y_OFFSET THEN
		temp :=cart_space - (posArrY[inc]-Y_OFFSET);
		posArrX[inc+1]:= temp+X_OFFSET;
		posArrY[inc+1]:= 0+Y_OFFSET;
		state:=1;
	ELSE
		posArrX[inc+1]:= 0+X_OFFSET;
		posArrY[inc+1]:=posArrY[inc]- cart_space;
		inc :=inc+1;
	END_IF
END_WHILE
inc := inc+1;

WHILE state = 1 DO // top
	IF posArrX[inc]+cart_space > (X_OFFSET+conv_length) THEN
		temp :=cart_space - ((X_OFFSET+conv_length)-posArrX[inc]);
		posArrX[inc+1]:= conv_length+X_OFFSET;
		posArrY[inc+1]:= temp+Y_OFFSET;
		state:=2;
	ELSE
		posArrX[inc+1]:= posArrX[inc]+cart_space;
		posArrY[inc+1]:=Y_OFFSET;
		inc :=inc+1;
	END_IF
END_WHILE
inc :=inc+1;	

WHILE state = 2 DO // right
	IF posArrY[inc]+cart_space > (Y_OFFSET+conv_height) THEN
		temp :=cart_space - ((Y_OFFSET+conv_height)-posArrY[inc]);
		posArrX[inc+1]:= (conv_length+X_OFFSET)-temp;
		posArrY[inc+1]:= 0+Y_OFFSET+conv_height;
		state:=3;
	ELSE
		posArrX[inc+1]:= 0+X_OFFSET+conv_length;
		posArrY[inc+1]:=posArrY[inc]+ cart_space;
		inc :=inc+1;
	END_IF	
END_WHILE
inc :=inc+1;	

WHILE state = 3 DO //bottom
	IF  posArrX[inc]-cart_space < X_OFFSET THEN
		temp :=cart_space - (posArrX[inc]-X_OFFSET);
		posArrX[inc+1]:= X_OFFSET;
		posArrY[inc+1]:= Y_OFFSET+ conv_height-temp;
		state:=4;
	ELSE
		posArrX[inc+1]:= posArrX[inc]-cart_space;
		posArrY[inc+1]:=Y_OFFSET+conv_height;
		inc :=inc+1;
		
	END_IF
END_WHILE

IF inc > 34 THEN
	RETURN;
END_IF


inc :=inc+1;

WHILE state = 4 DO    //left2
	IF posArrY[inc]-cart_space < ((conv_height/2)+Y_OFFSET) THEN
		state:=5;
	ELSE
		posArrX[inc+1]:= 0+X_OFFSET;
		posArrY[inc+1]:=posArrY[inc]- cart_space;
		inc :=inc+1;
		
	END_IF
END_WHILE
END_ACTION

ACTION A_SETUP:
bSTARTUP:=TRUE;
	fbCART[1].stCART.position:=1;
	fbCART[1].stCART.color:=1;
	fbCART[1].stCART.o_color:=1;
	fbCART[1].stCART.nNAME:=INT_TO_STRING(1001);
	fbCART[1].stCART.posX:=posArrX[1];
	fbCART[1].stCART.posY:=posArrY[1];
		
	FOR counter:=1 TO (num_of_carts-1) BY 1 DO
		fbCART[counter+1].stCART.position:=37-((counter*2));
		fbCART[counter+1].stCART.color:=1;
		fbCART[counter+1].stCART.o_color:=1;
		fbCART[counter+1].stCART.nNAME:=INT_TO_STRING(1000+counter+1);
		fbCART[counter+1].stCART.posX:=posArrX[37-((counter*2))];
		fbCART[counter+1].stCART.posY:=posArrY[37-((counter*2))];
	END_FOR;
END_ACTION

END_FUNCTION_BLOCK

// ---- STATIONS/FB_SUPPLY_CONV.TcPOU
FUNCTION_BLOCK FB_SUPPLY_CONV EXTENDS FB_STATION
VAR_INPUT
	fbAxis:REFERENCE TO FB_Axis;
END_VAR
VAR_OUTPUT
END_VAR
VAR
	rtrig_ERROR: R_TRIG;
END_VAR

CASE eSUPPLY_CONVAYOR_STATE OF
	E_CONVAYOR_STATE.homing:
		bHomed:=TRUE;
		eSUPPLY_CONVAYOR_STATE:=E_CONVAYOR_STATE.idle;
		fbAxis.bEnable:=TRUE;
		
	E_CONVAYOR_STATE.uninit:
		IF NOT bHomed THEN
			eSUPPLY_CONVAYOR_STATE:=E_CONVAYOR_STATE.homing;
		ELSE
			fbAxis.bMoveRel:=FALSE;
			fbAxis.bHalt:=FALSE;
			fbAxis.bReset:=FALSE;
			eSUPPLY_CONVAYOR_STATE:=E_CONVAYOR_STATE.idle;
		END_IF
		fbAxis.bDo_Step_FW:=FALSE;
		fbAxis.bMoveRel:=FALSE;
		fbAxis.stepFW_state:=0;
		fbAxis.bHalt:=FALSE;
		fbAxis.bReset:=FALSE;
		E_CONVAYOR_STATE.idle:
		
		//idle
	
	E_CONVAYOR_STATE.do_move: // start motion
		IF NOT fbAxis.bBusy  AND NOT fbAxis.bError THEN
			fbAxis.rPos:=0;	
			fbAxis.bSetPosition:=TRUE;	 
			fbAxis.bDo_Step_FW:=TRUE;
			eSUPPLY_CONVAYOR_STATE:=E_CONVAYOR_STATE.st1;
		END_IF
		
	E_CONVAYOR_STATE.st1:
		fbAxis.bDo_Step_FW:=FALSE;
		fbAxis.bSetPosition:=FALSE;
		eSUPPLY_CONVAYOR_STATE:=E_CONVAYOR_STATE.st2;	

	E_CONVAYOR_STATE.st2:
		IF fbAxis.bInPos THEN
			eSUPPLY_CONVAYOR_STATE:=E_CONVAYOR_STATE.done;
		END_IF
		
	E_CONVAYOR_STATE.done:
		//...
	
	E_CONVAYOR_STATE.pause:
	//paused
	
	E_CONVAYOR_STATE.estop:
		fbAxis.bHalt:=TRUE;
		fbAxis.bReset:=TRUE;
		bHomed:=FALSE;
	
	E_CONVAYOR_STATE.error:
		//...
		
	rtrig_ERROR(CLK:=(eSUPPLY_CONVAYOR_STATE=E_CONVAYOR_STATE.error), Q=> );
	IF rtrig_ERROR.Q THEN
		gEventType:= 'Alarm'; 
		gEventSeverity:= 'Error';
		gEventIdentity:=3001;
		gEventName:= 'SUPPLY CONVAYOR';
		gEventText:='MOTOR ERROR:';
		fbEventLogger.mAdd();
	END_IF
END_CASE

END_FUNCTION_BLOCK

// ---- Functions/F_Linear.TcPOU
FUNCTION F_Linear : real
VAR_INPUT
	analog_read:INT;
	IO_min, IO_max, eng_min, eng_max:REAL;
END_VAR
VAR
END_VAR

IF  (IO_max - IO_min) > 0 THEN
	F_linear :=  ((eng_max - eng_min)/(IO_max - IO_min))*(analog_read - IO_max) + eng_max;
ELSE
	F_linear :=  0;
END_IF

END_FUNCTION

// ---- POUs/prg_CSV_V2.TcPOU
PROGRAM prg_CSV_V2
VAR
	FilePathAndName: STRING:='C:\temp\Records_X-X-XX.xls';// Path for Win CE: 'Hard Disk\ftp\Records_X-X-XX.xls';
	
	fbFileOpen					:	FB_FileOpen;
	fbFileClose					:	FB_FileClose;
	fbFileWrite					:	FB_FileWrite;
	fbFileGet					:	FB_FileGets;
	
	bFirstCycle:BOOL:=TRUE;//:=TRUE;	
	bWrite: BOOL;
	bStart: BOOL;
	iState: INT;
	hFile: UINT;
	i:INT:=1;

	bBusy: BOOL;
	bDone: BOOL;
	bError: BOOL;

	sLine: STRING;
	sLineToWrite:STRING(255);
	sHeader :STRING(255):='Time Stamp$TDescription$TValu$TUnit';
	iErrorState: INT;
	FirstLine: STRING;


	
//Data to Write
	arrDataToWrite:ARRAY[1..C_MaxParametersToWrite]OF ST_CsvTableRowData;
	tonPulseGenerator:ton;
	
//get System Time ( for CSV time stamp )	
	fbLocalSystemTime:FB_LocalSystemTime;
	tonWritingCyclie:ton;
	sSyatemTime: STRING(24);
	wDayMem:WORD;
	
	
END_VAR
VAR CONSTANT
	C_MaxParametersToWrite:INT:=1;
END_VAR

//get System Time ( for CSV time stamp )
fbLocalSystemTime( bEnable:= TRUE ); 
sSyatemTime:=SYSTEMTIME_TO_STRING(fbLocalSystemTime.systemTime);

//Set data to write
	//Analog data 1
	arrDataToWrite[1].sTimeStamp:=sSyatemTime;
	arrDataToWrite[1].sType:=gEventType;
	arrDataToWrite[1].sSeverity:=gEventSeverity;
	arrDataToWrite[1].sIdentity:=UDINT_TO_STRING(gEventIdentity);
	arrDataToWrite[1].sName:=gEventName;
	arrDataToWrite[1].sText:=gEventText;
	arrDataToWrite[1].sP_CAPSULE :=LREAL_TO_STRING(0);
	arrDataToWrite[1].sSel_FEED :=LREAL_TO_STRING(0);
	arrDataToWrite[1].sSel_PRODUCT :=LREAL_TO_STRING(0);
	arrDataToWrite[1].sUnit :=LREAL_TO_STRING(0);
	
	//Analog data 2
	//arrDataToWrite[2].sDescription:='Humidity sensor 2';
	//arrDataToWrite[2].sUnit:='%';
	//arrDataToWrite[2].sTimeStamp:=sSyatemTime;
	//arrDataToWrite[2].sValue:=REAL_TO_STRING(2);
	
    

//Writing rate
tonWritingCyclie(IN:= NOT tonWritingCyclie.Q , PT:= T#30S , Q=> , ET=> );
IF WriteLogToFile THEN
	WriteLogToFile:=FALSE;
	//Create new file every day
	IF wDayMem <> fbLocalSystemTime.systemTime.wDay OR bFirstCycle  THEN
			wDayMem:=fbLocalSystemTime.systemTime.wDay;
			FilePathAndName:=concat('C:\LOGS\TAMAR',concat('-',concat(WORD_TO_STRING(fbLocalSystemTime.systemTime.wDay),concat('-',concat(WORD_TO_STRING(fbLocalSystemTime.systemTime.wMonth),concat('-',concat(WORD_TO_STRING(fbLocalSystemTime.systemTime.wYear),'.xls')))))));
			bFirstCycle:=FALSE;
	END_IF
	bWrite:=TRUE;
END_IF	

//Excel coloms Header
sHeader:='Time Stamp$TTYPE$TSEVERITY$TIDENTITY$TNAME$TTEXT$T$T$T$T';


CASE iState OF
	0:	IF bWrite THEN
			fbFileOpen.bExecute := FALSE;
			fbFileClose.bExecute := FALSE;
			fbFileWrite.bExecute := FALSE;
			fbFileGet.bExecute := FALSE;
			bDone:=FALSE;
			bError:=FALSE;
			bWrite:=FALSE;
			iState := iState + 1;
		END_IF

	1:	(* open a file to test it's content *)
		fbFileOpen(
			sPathName:=FilePathAndName ,
			nMode:= FOPEN_MODEAPPEND OR FOPEN_MODEPLUS OR FOPEN_MODETEXT ,
			bExecute:=TRUE  );
	
		IF fbFileOpen.bBusy THEN
			iState := iState + 1;
		END_IF

	2:	IF NOT fbFileOpen.bBusy AND NOT fbFileOpen.bError THEN
			hFile:=fbFileOpen.hFile;
			fbFileOpen.bExecute := FALSE;
			iState := iState + 1;
		ELSIF fbFileOpen.bError THEN
			iErrorState:=iState;
			iState := 99;
		END_IF


	3:	(*Get First line to check if file allready writen *)
		fbFileGet(
			hFile:=hFile ,
			bExecute:=TRUE ,
			tTimeout:=T#1s ,
			sLine=>FirstLine ,
			bEOF=> );

		IF fbFileGet.bBusy THEN
			iState := iState + 1;
		END_IF;

	4:	IF NOT fbFileGet.bBusy AND NOT fbFileGet.bError THEN
			fbFileGet(bExecute:=FALSE);
			IF FirstLine='' THEN
				iState := iState + 1;
			ELSE
				iState:=10;
			END_IF
		ELSIF fbFileGet.bError THEN
			iErrorState:=iState;
			iState := 99;
		END_IF


	5:	(*write file header*)
		fbFileWrite(
				sNetId:='' ,
				hFile:=hFile ,
				pWriteBuff:= ADR(sHeader),
				cbWriteLen:=INT_TO_UDINT (LEN(sHeader)) ,
				bExecute:=TRUE ,
				tTimeout:=T#5s );

		IF fbFileWrite.bBusy THEN
			iState := iState + 1;
		END_IF;


	6:	IF  NOT fbFileWrite.bBusy
			AND NOT fbFileWrite.bError   THEN
				fbFileWrite.bExecute:=FALSE;
				iState := iState + 1;
		ELSIF fbFileWrite.bError THEN
			iErrorState:=iState;
			iState := 99;
		END_IF


	7: (*close the file handle*)
		fbFileClose.bExecute := TRUE;
		fbFileClose.hFile := hFile;
		IF fbFileClose.bBusy THEN
			iState := iState + 1;
		END_IF;

	8:	IF NOT fbFileClose.bBusy AND NOT fbFileClose.bError THEN
			fbFileClose.bExecute := FALSE;
			iState := 10;
		ELSIF fbFileClose.bError THEN
			iErrorState:=iState;
			iState := 99;
		END_IF

	10:	(* open a file to append line*)
		fbFileOpen(
			sPathName:=FilePathAndName ,
			nMode:= FOPEN_MODEAPPEND ,
			bExecute:=TRUE ,
			hFile=>hFile );
	
		IF fbFileOpen.bBusy THEN
			iState := iState + 1;
		END_IF

	11:	IF NOT fbFileOpen.bBusy AND NOT fbFileOpen.bError THEN
			hFile:=fbFileOpen.hFile;
			fbFileOpen.bExecute := FALSE;
			iState := iState + 4;
		ELSIF fbFileOpen.bError THEN
			iErrorState:=iState;
			iState := 99;
		END_IF



	15:	(* write data into log file*)
		IF i > 0 AND i <= C_MaxParametersToWrite THEN
			sLineToWrite:=CONCAT('$N',
				concat(sSyatemTime,
					concat('$T',
						concat(arrDataToWrite[i].sType,
							concat('$T',
								concat(arrDataToWrite[i].sSeverity,
									concat('$T',
										concat(arrDataToWrite[i].sIdentity,
											concat('$T',
												concat(arrDataToWrite[i].sName,
													concat('$T',
														concat(arrDataToWrite[i].sText,
															concat('$T',
																concat(arrDataToWrite[i].sSel_FEED,
																		concat('$T',
																			concat(arrDataToWrite[i].sSel_PRODUCT,
																				concat('$T',
																					concat(arrDataToWrite[i].sP_TRANSFER,
																						concat('$T',
																							concat(arrDataToWrite[i].sP_CAPSULE,
																								concat('$T',arrDataToWrite[i].sUnit)))))))))))))))))))));
			sLog:=sLineToWrite;// copy string to GVL string
			fbFileWrite(
				sNetId:='' ,
				hFile:=hFile ,
				pWriteBuff:= ADR(sLineToWrite),
				cbWriteLen:=INT_TO_UDINT (LEN(sLineToWrite)) ,
				bExecute:=TRUE ,
				tTimeout:=T#10S ,
				bBusy=> ,
				bError=>,
				nErrId=> );

		ELSE
			iState:=80;
		END_IF

		

		IF  NOT fbFileWrite.bBusy
			AND NOT fbFileWrite.bError   THEN
			fbFileWrite.bExecute:=FALSE;
			i:=i+1;
			//iState:=80;
		END_IF


	80: (*close the file handle*)
		i:=1;
		fbFileClose.bExecute := TRUE;
		fbFileClose.hFile := hFile;
		IF fbFileClose.bBusy THEN
			iState := iState + 1;
		END_IF;

	81:	IF NOT fbFileClose.bBusy AND NOT fbFileClose.bError THEN
			fbFileClose.bExecute := FALSE;
			iState := 88;
			hFile := fbFileClose.hFile;
		ELSIF fbFileClose.bError THEN
			iErrorState:=iState;
			iState := 99;
		END_IF

	88: bBusy := FALSE;
		bDone := NOT bError;
		iState := 0;
		i:=1;

	99:	bError := TRUE;
		iState := 88;

END_CASE;
fbFileOpen();
fbFileClose();
fbFileWrite();
fbFileGet();

END_PROGRAM

// ---- POUs/MOTORS.TcPOU
PROGRAM MOTORS
VAR
	
END_VAR

Axis_MAIN(sName:='MAIN');
Axis_SUPPLY(sNAme:='SUPPLY');
Axis_JACK1(sNAme:='JACK1');
Axis_JACK2(sNAme:='JACK2');

END_PROGRAM

// ---- POUs/PISTONS/PIST_CYCLE.TcPOU
PROGRAM PIST_CYCLE
VAR
	bFirstRun:BOOL:=FALSE;
	counter :INT;
END_VAR


IF NOT bFirstRun THEN
	FOR counter:=1 TO iNUMBER_OF_PISTONS BY 1 DO
		fbPist[counter].bInit:=1;
	END_FOR;
bFirstRun:=TRUE;
END_IF
 

feeder();
clean();
extract();
drop();
separate1();
separate2();

ACTION clean:
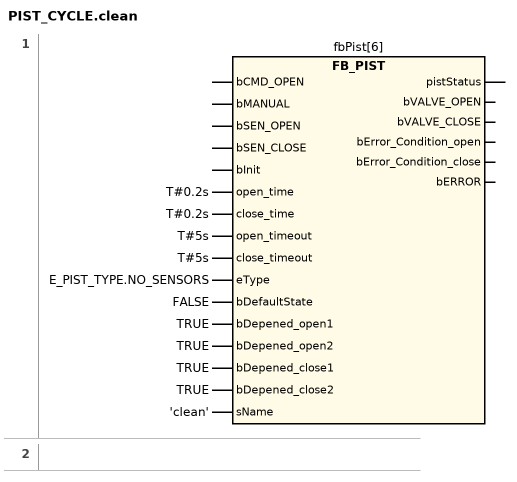
// NETWORK 1
fbPist[6](
    open_time := T#0.2s,
    close_time := T#0.2s,
    open_timeout := T#5s,
    close_timeout := T#5s,
    eType := E_PIST_TYPE.NO_SENSORS,
    bDefaultState := FALSE,
    bDepened_open1 := TRUE,
    bDepened_open2 := TRUE,
    bDepened_close1 := TRUE,
    bDepened_close2 := TRUE,
    sName := 'clean'); // FB_PIST

// NETWORK 2
END_ACTION

ACTION drop:
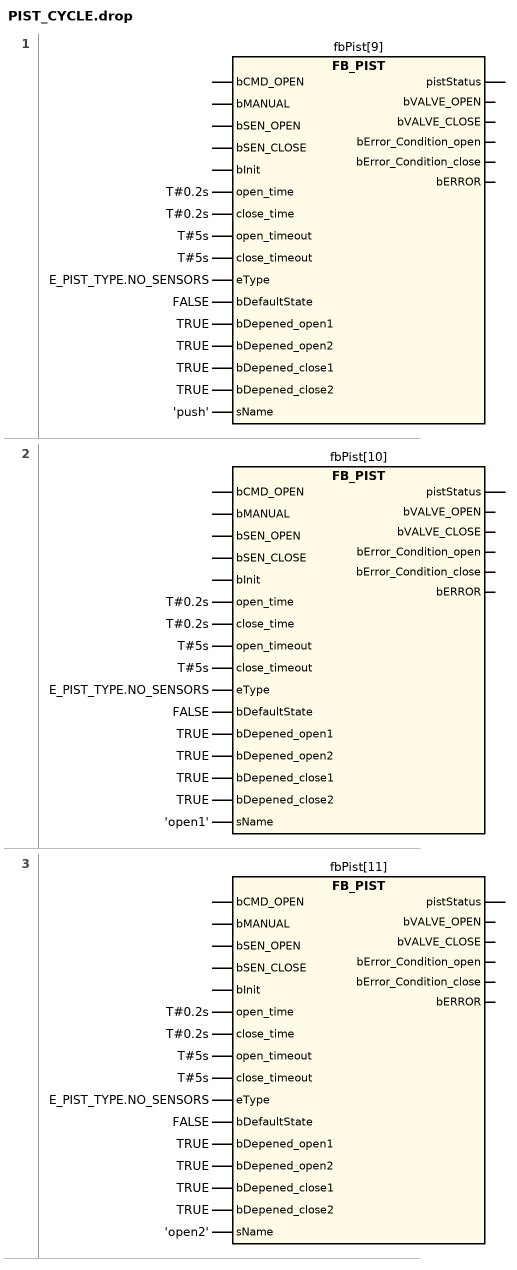
// NETWORK 1
fbPist[9](
    open_time := T#0.2s,
    close_time := T#0.2s,
    open_timeout := T#5s,
    close_timeout := T#5s,
    eType := E_PIST_TYPE.NO_SENSORS,
    bDefaultState := FALSE,
    bDepened_open1 := TRUE,
    bDepened_open2 := TRUE,
    bDepened_close1 := TRUE,
    bDepened_close2 := TRUE,
    sName := 'push'); // FB_PIST

// NETWORK 2
fbPist[10](
    open_time := T#0.2s,
    close_time := T#0.2s,
    open_timeout := T#5s,
    close_timeout := T#5s,
    eType := E_PIST_TYPE.NO_SENSORS,
    bDefaultState := FALSE,
    bDepened_open1 := TRUE,
    bDepened_open2 := TRUE,
    bDepened_close1 := TRUE,
    bDepened_close2 := TRUE,
    sName := 'open1'); // FB_PIST

// NETWORK 3
fbPist[11](
    open_time := T#0.2s,
    close_time := T#0.2s,
    open_timeout := T#5s,
    close_timeout := T#5s,
    eType := E_PIST_TYPE.NO_SENSORS,
    bDefaultState := FALSE,
    bDepened_open1 := TRUE,
    bDepened_open2 := TRUE,
    bDepened_close1 := TRUE,
    bDepened_close2 := TRUE,
    sName := 'open2'); // FB_PIST
END_ACTION

ACTION extract:
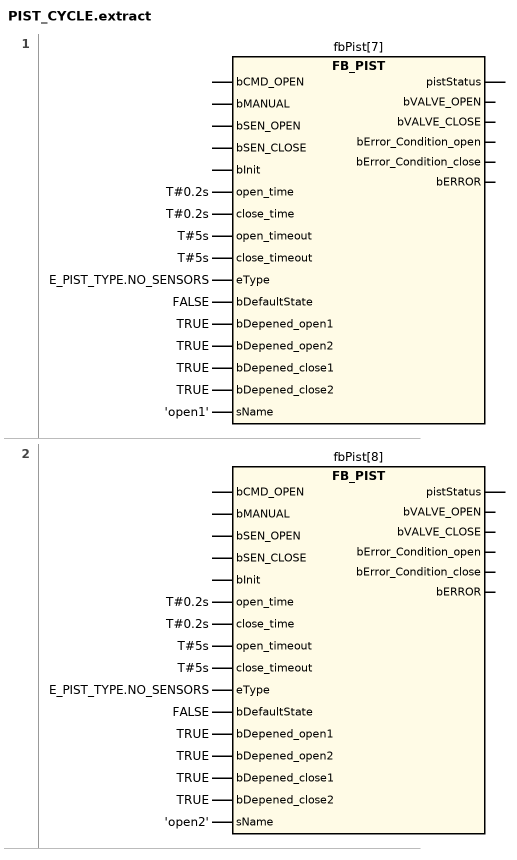
// NETWORK 1
fbPist[7](
    open_time := T#0.2s,
    close_time := T#0.2s,
    open_timeout := T#5s,
    close_timeout := T#5s,
    eType := E_PIST_TYPE.NO_SENSORS,
    bDefaultState := FALSE,
    bDepened_open1 := TRUE,
    bDepened_open2 := TRUE,
    bDepened_close1 := TRUE,
    bDepened_close2 := TRUE,
    sName := 'open1'); // FB_PIST

// NETWORK 2
fbPist[8](
    open_time := T#0.2s,
    close_time := T#0.2s,
    open_timeout := T#5s,
    close_timeout := T#5s,
    eType := E_PIST_TYPE.NO_SENSORS,
    bDefaultState := FALSE,
    bDepened_open1 := TRUE,
    bDepened_open2 := TRUE,
    bDepened_close1 := TRUE,
    bDepened_close2 := TRUE,
    sName := 'open2'); // FB_PIST
END_ACTION

ACTION feeder:
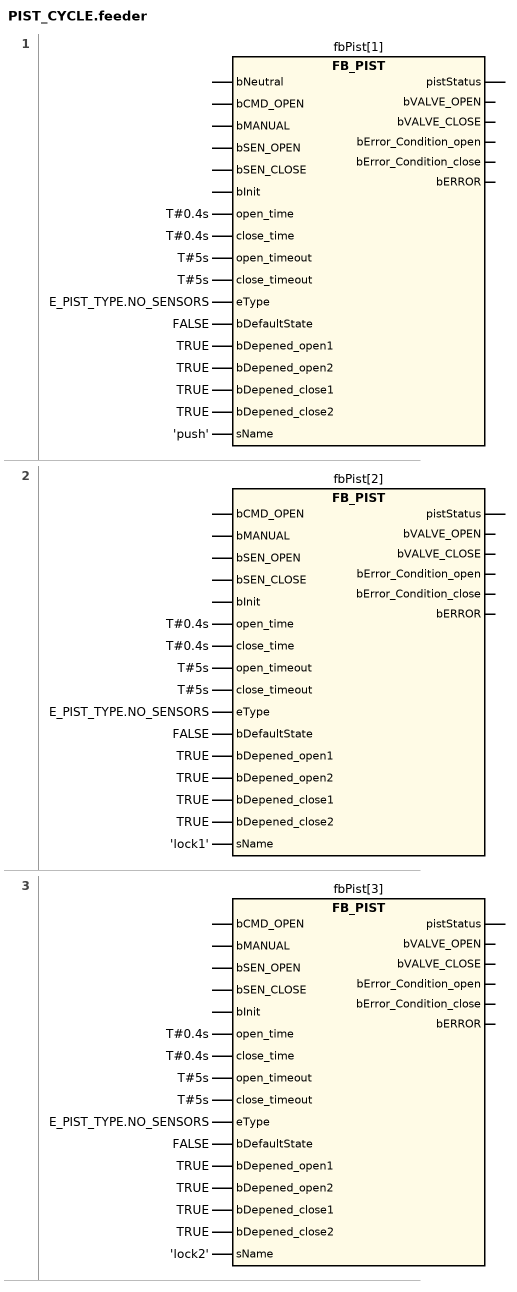
// NETWORK 1
fbPist[1](
    open_time := T#0.4s,
    close_time := T#0.4s,
    open_timeout := T#5s,
    close_timeout := T#5s,
    eType := E_PIST_TYPE.NO_SENSORS,
    bDefaultState := FALSE,
    bDepened_open1 := TRUE,
    bDepened_open2 := TRUE,
    bDepened_close1 := TRUE,
    bDepened_close2 := TRUE,
    sName := 'push'); // FB_PIST

// NETWORK 2
fbPist[2](
    open_time := T#0.4s,
    close_time := T#0.4s,
    open_timeout := T#5s,
    close_timeout := T#5s,
    eType := E_PIST_TYPE.NO_SENSORS,
    bDefaultState := FALSE,
    bDepened_open1 := TRUE,
    bDepened_open2 := TRUE,
    bDepened_close1 := TRUE,
    bDepened_close2 := TRUE,
    sName := 'lock1'); // FB_PIST

// NETWORK 3
fbPist[3](
    open_time := T#0.4s,
    close_time := T#0.4s,
    open_timeout := T#5s,
    close_timeout := T#5s,
    eType := E_PIST_TYPE.NO_SENSORS,
    bDefaultState := FALSE,
    bDepened_open1 := TRUE,
    bDepened_open2 := TRUE,
    bDepened_close1 := TRUE,
    bDepened_close2 := TRUE,
    sName := 'lock2'); // FB_PIST

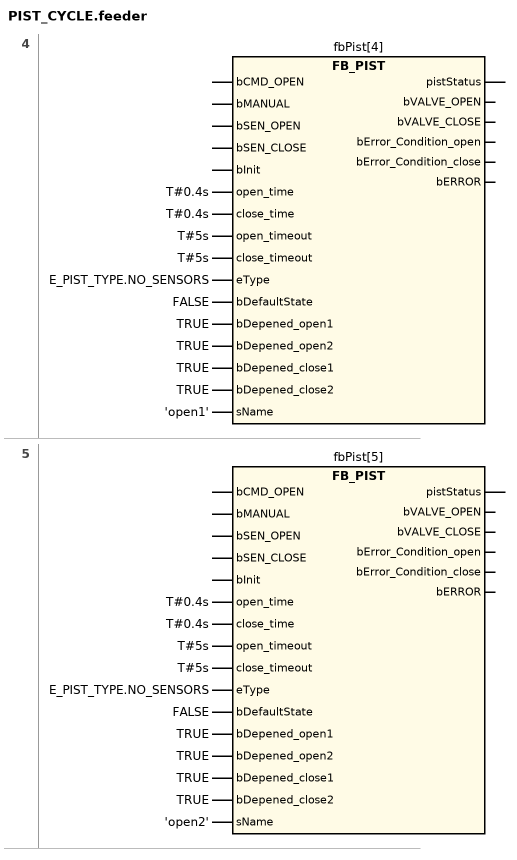
// NETWORK 4
fbPist[4](
    open_time := T#0.4s,
    close_time := T#0.4s,
    open_timeout := T#5s,
    close_timeout := T#5s,
    eType := E_PIST_TYPE.NO_SENSORS,
    bDefaultState := FALSE,
    bDepened_open1 := TRUE,
    bDepened_open2 := TRUE,
    bDepened_close1 := TRUE,
    bDepened_close2 := TRUE,
    sName := 'open1'); // FB_PIST

// NETWORK 5
fbPist[5](
    open_time := T#0.4s,
    close_time := T#0.4s,
    open_timeout := T#5s,
    close_timeout := T#5s,
    eType := E_PIST_TYPE.NO_SENSORS,
    bDefaultState := FALSE,
    bDepened_open1 := TRUE,
    bDepened_open2 := TRUE,
    bDepened_close1 := TRUE,
    bDepened_close2 := TRUE,
    sName := 'open2'); // FB_PIST
END_ACTION

ACTION separate1:
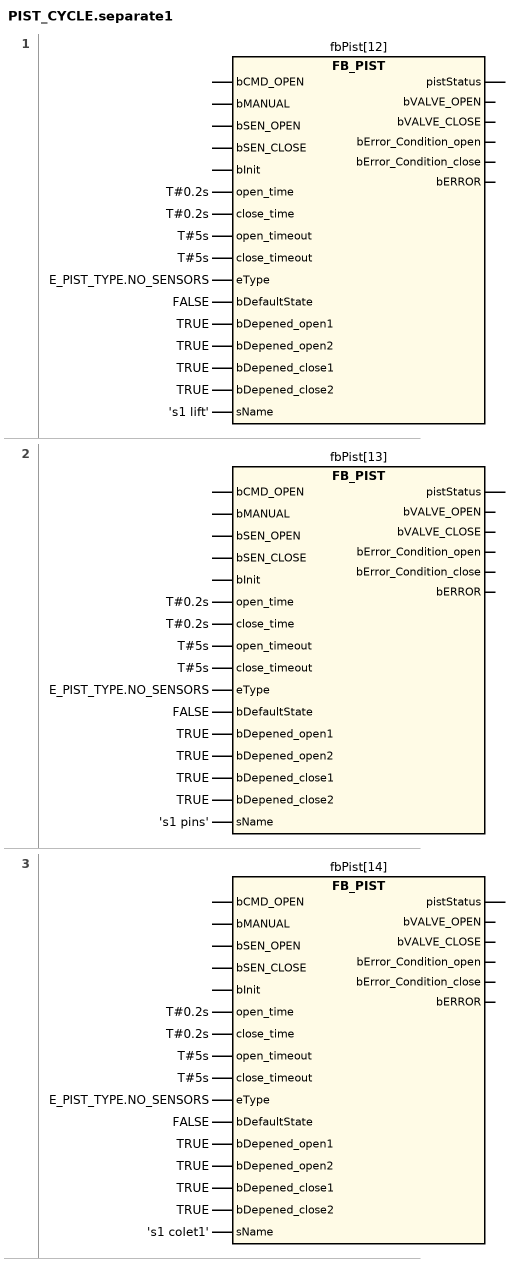
// NETWORK 1
fbPist[12](
    open_time := T#0.2s,
    close_time := T#0.2s,
    open_timeout := T#5s,
    close_timeout := T#5s,
    eType := E_PIST_TYPE.NO_SENSORS,
    bDefaultState := FALSE,
    bDepened_open1 := TRUE,
    bDepened_open2 := TRUE,
    bDepened_close1 := TRUE,
    bDepened_close2 := TRUE,
    sName := 's1 lift'); // FB_PIST

// NETWORK 2
fbPist[13](
    open_time := T#0.2s,
    close_time := T#0.2s,
    open_timeout := T#5s,
    close_timeout := T#5s,
    eType := E_PIST_TYPE.NO_SENSORS,
    bDefaultState := FALSE,
    bDepened_open1 := TRUE,
    bDepened_open2 := TRUE,
    bDepened_close1 := TRUE,
    bDepened_close2 := TRUE,
    sName := 's1 pins'); // FB_PIST

// NETWORK 3
fbPist[14](
    open_time := T#0.2s,
    close_time := T#0.2s,
    open_timeout := T#5s,
    close_timeout := T#5s,
    eType := E_PIST_TYPE.NO_SENSORS,
    bDefaultState := FALSE,
    bDepened_open1 := TRUE,
    bDepened_open2 := TRUE,
    bDepened_close1 := TRUE,
    bDepened_close2 := TRUE,
    sName := 's1 colet1'); // FB_PIST

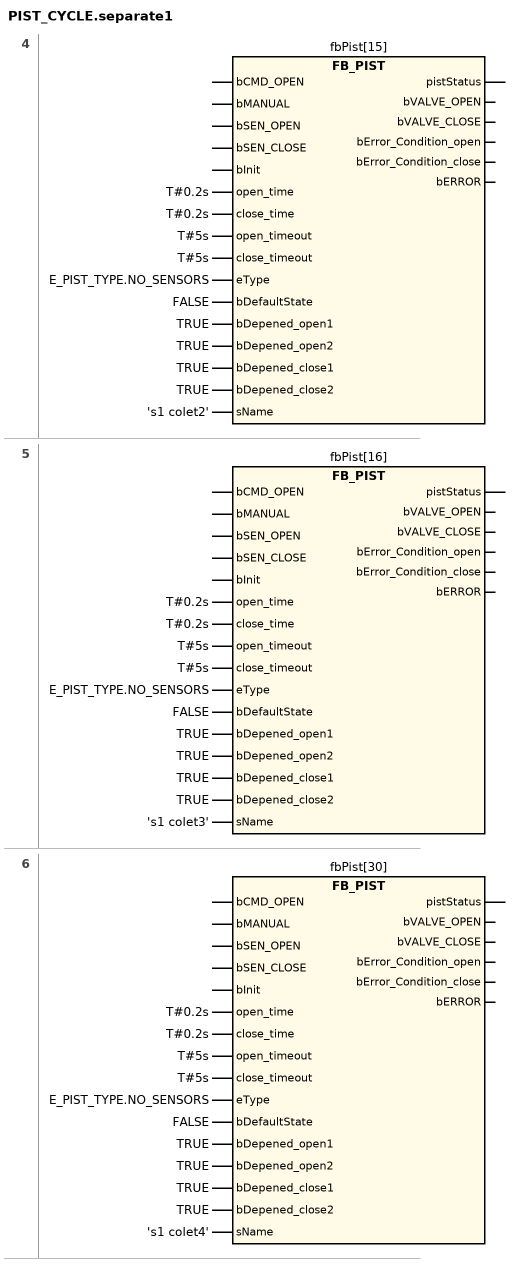
// NETWORK 4
fbPist[15](
    open_time := T#0.2s,
    close_time := T#0.2s,
    open_timeout := T#5s,
    close_timeout := T#5s,
    eType := E_PIST_TYPE.NO_SENSORS,
    bDefaultState := FALSE,
    bDepened_open1 := TRUE,
    bDepened_open2 := TRUE,
    bDepened_close1 := TRUE,
    bDepened_close2 := TRUE,
    sName := 's1 colet2'); // FB_PIST

// NETWORK 5
fbPist[16](
    open_time := T#0.2s,
    close_time := T#0.2s,
    open_timeout := T#5s,
    close_timeout := T#5s,
    eType := E_PIST_TYPE.NO_SENSORS,
    bDefaultState := FALSE,
    bDepened_open1 := TRUE,
    bDepened_open2 := TRUE,
    bDepened_close1 := TRUE,
    bDepened_close2 := TRUE,
    sName := 's1 colet3'); // FB_PIST

// NETWORK 6
fbPist[30](
    open_time := T#0.2s,
    close_time := T#0.2s,
    open_timeout := T#5s,
    close_timeout := T#5s,
    eType := E_PIST_TYPE.NO_SENSORS,
    bDefaultState := FALSE,
    bDepened_open1 := TRUE,
    bDepened_open2 := TRUE,
    bDepened_close1 := TRUE,
    bDepened_close2 := TRUE,
    sName := 's1 colet4'); // FB_PIST

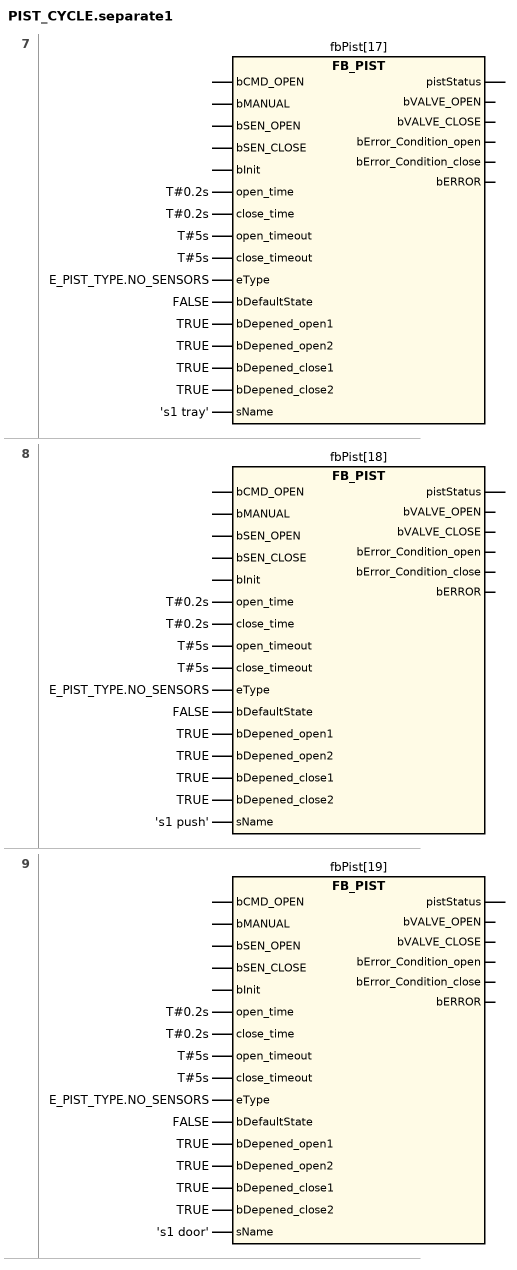
// NETWORK 7
fbPist[17](
    open_time := T#0.2s,
    close_time := T#0.2s,
    open_timeout := T#5s,
    close_timeout := T#5s,
    eType := E_PIST_TYPE.NO_SENSORS,
    bDefaultState := FALSE,
    bDepened_open1 := TRUE,
    bDepened_open2 := TRUE,
    bDepened_close1 := TRUE,
    bDepened_close2 := TRUE,
    sName := 's1 tray'); // FB_PIST

// NETWORK 8
fbPist[18](
    open_time := T#0.2s,
    close_time := T#0.2s,
    open_timeout := T#5s,
    close_timeout := T#5s,
    eType := E_PIST_TYPE.NO_SENSORS,
    bDefaultState := FALSE,
    bDepened_open1 := TRUE,
    bDepened_open2 := TRUE,
    bDepened_close1 := TRUE,
    bDepened_close2 := TRUE,
    sName := 's1 push'); // FB_PIST

// NETWORK 9
fbPist[19](
    open_time := T#0.2s,
    close_time := T#0.2s,
    open_timeout := T#5s,
    close_timeout := T#5s,
    eType := E_PIST_TYPE.NO_SENSORS,
    bDefaultState := FALSE,
    bDepened_open1 := TRUE,
    bDepened_open2 := TRUE,
    bDepened_close1 := TRUE,
    bDepened_close2 := TRUE,
    sName := 's1 door'); // FB_PIST
END_ACTION

ACTION separate2:
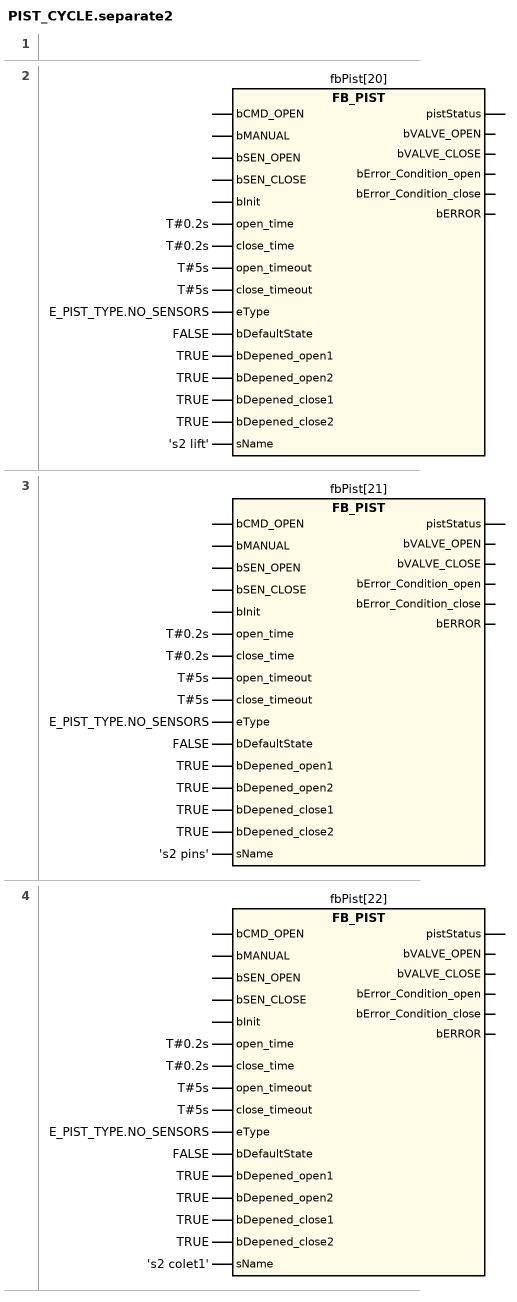
// NETWORK 1

// NETWORK 2
fbPist[20](
    open_time := T#0.2s,
    close_time := T#0.2s,
    open_timeout := T#5s,
    close_timeout := T#5s,
    eType := E_PIST_TYPE.NO_SENSORS,
    bDefaultState := FALSE,
    bDepened_open1 := TRUE,
    bDepened_open2 := TRUE,
    bDepened_close1 := TRUE,
    bDepened_close2 := TRUE,
    sName := 's2 lift'); // FB_PIST

// NETWORK 3
fbPist[21](
    open_time := T#0.2s,
    close_time := T#0.2s,
    open_timeout := T#5s,
    close_timeout := T#5s,
    eType := E_PIST_TYPE.NO_SENSORS,
    bDefaultState := FALSE,
    bDepened_open1 := TRUE,
    bDepened_open2 := TRUE,
    bDepened_close1 := TRUE,
    bDepened_close2 := TRUE,
    sName := 's2 pins'); // FB_PIST

// NETWORK 4
fbPist[22](
    open_time := T#0.2s,
    close_time := T#0.2s,
    open_timeout := T#5s,
    close_timeout := T#5s,
    eType := E_PIST_TYPE.NO_SENSORS,
    bDefaultState := FALSE,
    bDepened_open1 := TRUE,
    bDepened_open2 := TRUE,
    bDepened_close1 := TRUE,
    bDepened_close2 := TRUE,
    sName := 's2 colet1'); // FB_PIST

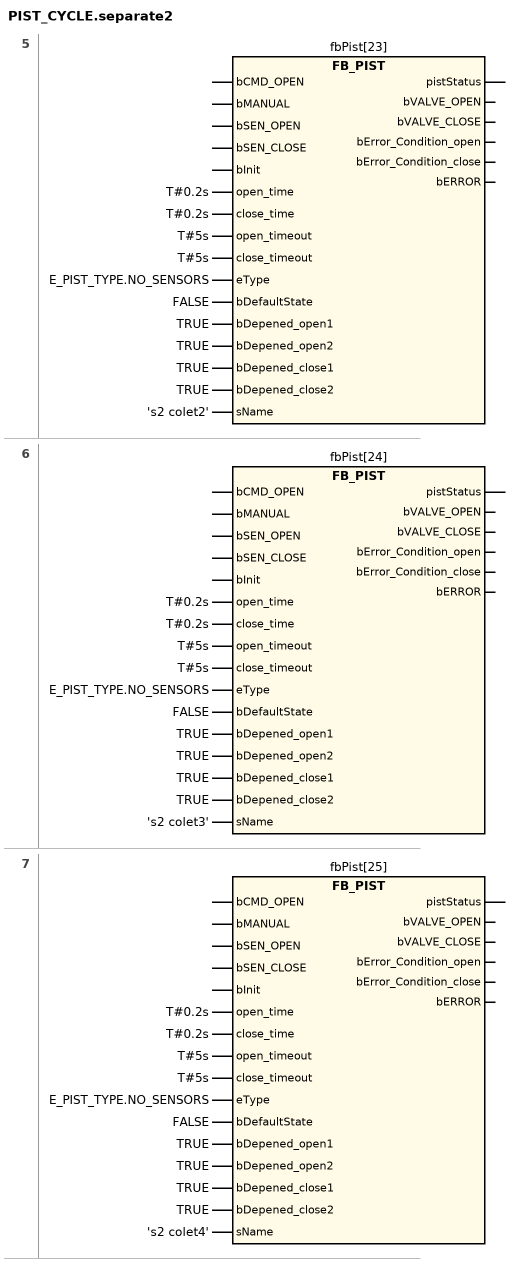
// NETWORK 5
fbPist[23](
    open_time := T#0.2s,
    close_time := T#0.2s,
    open_timeout := T#5s,
    close_timeout := T#5s,
    eType := E_PIST_TYPE.NO_SENSORS,
    bDefaultState := FALSE,
    bDepened_open1 := TRUE,
    bDepened_open2 := TRUE,
    bDepened_close1 := TRUE,
    bDepened_close2 := TRUE,
    sName := 's2 colet2'); // FB_PIST

// NETWORK 6
fbPist[24](
    open_time := T#0.2s,
    close_time := T#0.2s,
    open_timeout := T#5s,
    close_timeout := T#5s,
    eType := E_PIST_TYPE.NO_SENSORS,
    bDefaultState := FALSE,
    bDepened_open1 := TRUE,
    bDepened_open2 := TRUE,
    bDepened_close1 := TRUE,
    bDepened_close2 := TRUE,
    sName := 's2 colet3'); // FB_PIST

// NETWORK 7
fbPist[25](
    open_time := T#0.2s,
    close_time := T#0.2s,
    open_timeout := T#5s,
    close_timeout := T#5s,
    eType := E_PIST_TYPE.NO_SENSORS,
    bDefaultState := FALSE,
    bDepened_open1 := TRUE,
    bDepened_open2 := TRUE,
    bDepened_close1 := TRUE,
    bDepened_close2 := TRUE,
    sName := 's2 colet4'); // FB_PIST

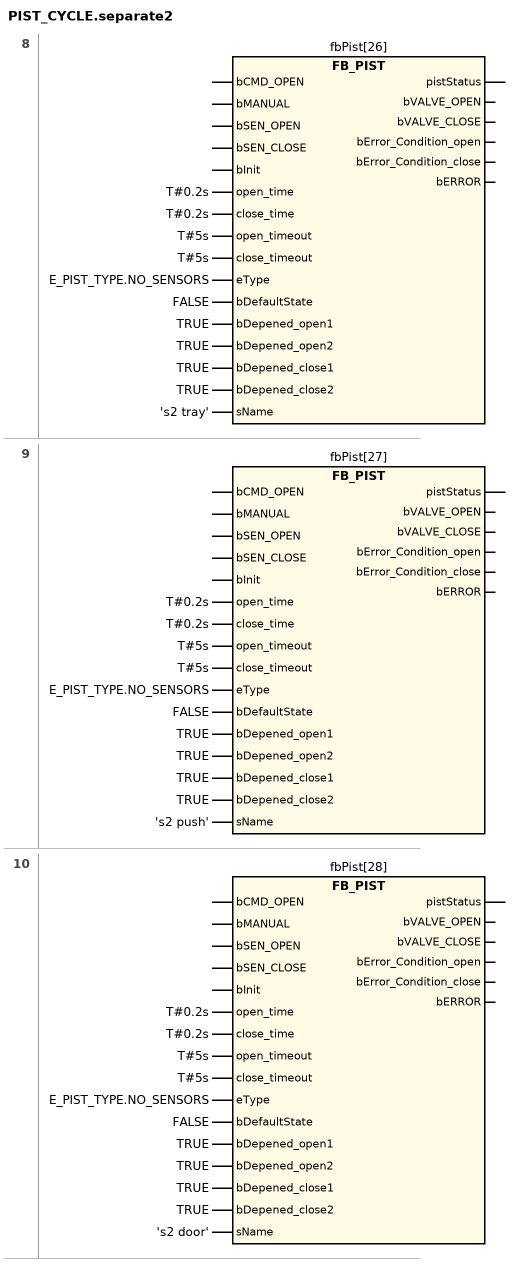
// NETWORK 8
fbPist[26](
    open_time := T#0.2s,
    close_time := T#0.2s,
    open_timeout := T#5s,
    close_timeout := T#5s,
    eType := E_PIST_TYPE.NO_SENSORS,
    bDefaultState := FALSE,
    bDepened_open1 := TRUE,
    bDepened_open2 := TRUE,
    bDepened_close1 := TRUE,
    bDepened_close2 := TRUE,
    sName := 's2 tray'); // FB_PIST

// NETWORK 9
fbPist[27](
    open_time := T#0.2s,
    close_time := T#0.2s,
    open_timeout := T#5s,
    close_timeout := T#5s,
    eType := E_PIST_TYPE.NO_SENSORS,
    bDefaultState := FALSE,
    bDepened_open1 := TRUE,
    bDepened_open2 := TRUE,
    bDepened_close1 := TRUE,
    bDepened_close2 := TRUE,
    sName := 's2 push'); // FB_PIST

// NETWORK 10
fbPist[28](
    open_time := T#0.2s,
    close_time := T#0.2s,
    open_timeout := T#5s,
    close_timeout := T#5s,
    eType := E_PIST_TYPE.NO_SENSORS,
    bDefaultState := FALSE,
    bDepened_open1 := TRUE,
    bDepened_open2 := TRUE,
    bDepened_close1 := TRUE,
    bDepened_close2 := TRUE,
    sName := 's2 door'); // FB_PIST
END_ACTION

END_PROGRAM

// ---- POUs/FB_EventLogger.TcPOU
FUNCTION_BLOCK FB_EventLogger
VAR_INPUT
END_VAR
VAR_OUTPUT
END_VAR
VAR
	buffer_counter:INT;
	EventBuffer: ARRAY[1..MAXIMUN_SIZE_OF_EVENT_BUFFR] OF ST_Event;
	EventBuffer_clear: ARRAY[1..MAXIMUN_SIZE_OF_EVENT_BUFFR] OF ST_Event;
	EventBufferIndex:INT:=0;
END_VAR
VAR CONSTANT
	MAXIMUN_SIZE_OF_EVENT_BUFFR:INT :=100;
END_VAR

METHOD IsEventBufferFull : BOOL
VAR_INPUT
END_VAR
IF (EventBufferIndex+1) > MAXIMUN_SIZE_OF_EVENT_BUFFR THEN
	EventBuffer:=EventBuffer_clear;
	EventBufferIndex:=0 ;
	//IsEventBufferFull:=TRUE; 
END_IF
IsEventBufferFull:=FALSE;
END_METHOD

(* returns false if not succesfull*) 
METHOD PUBLIC mAdd : BOOL
VAR_INPUT
	
END_VAR

VAR
	arrDataToWrite: INT;
END_VAR

IF NOT IsEventBufferFull() THEN
	EventBufferIndex:=EventBufferIndex+1;
	EventBuffer[EventBufferIndex].eEventType:=gEventType;
	EventBuffer[EventBufferIndex].eEventSeverity:=gEventSeverity;
	EventBuffer[EventBufferIndex].nEventIdentity:=gEventIdentity;
	EventBuffer[EventBufferIndex].sEventName:=gEventName;
	EventBuffer[EventBufferIndex].sEventText:=gEventText;
	UpdateEventTimestampWithSystemTime (stEvent:=EventBuffer[EventBufferIndex]); 
	sEventTime:= DT_TO_STRING (EventBuffer[EventBufferIndex].dtTimestamp);
	mAdd:=TRUE ;
ELSE
	mAdd:=FALSE;
END_IF
END_METHOD

END_FUNCTION_BLOCK

// ---- Functions/UpdateEventTimestampWithSystemTime.TcPOU
FUNCTION UpdateEventTimestampWithSystemTime 
VAR_INPUT
	stEvent: REFERENCE TO ST_Event;  
	
END_VAR
VAR
	fbGETSYSTEMTIME : GETSYSTEMTIME;
	stFileTime : T_FILETIME;
END_VAR

fbGETSYSTEMTIME(timeLoDW =>stFileTime.dwLowDateTime ,
				timeHiDW =>stFileTime.dwHighDateTime );
				
stEvent.dtTimestamp:= FILETIME_TO_DT(fileTime := stFileTime);

END_FUNCTION

// ---- Checks/CheckBounds.TcPOU
// Implicitly generated code : DO NOT EDIT
FUNCTION CheckBounds : DINT
VAR_INPUT
	index, lower, upper: DINT;
END_VAR

// Implicitly generated code : Only an Implementation suggestion
{noflow}
IF  index < lower THEN
	CheckBounds := lower;
ELSIF  index > upper THEN
	CheckBounds := upper;
ELSE  
	CheckBounds := index;
END_IF
{flow}

END_FUNCTION

// ---- Checks/CheckDivDInt.TcPOU
// Implicitly generated code : DO NOT EDIT
FUNCTION CheckDivDInt : DINT
VAR_INPUT
	divisor:DINT;
END_VAR

// Implicitly generated code : Only an Implementation suggestion
{noflow}
IF divisor = 0 THEN
	CheckDivDInt:=1;
ELSE
	CheckDivDInt:=divisor;
END_IF;
{flow}

END_FUNCTION

// ---- Checks/CheckDivLInt.TcPOU
// Implicitly generated code : DO NOT EDIT
FUNCTION CheckDivLInt : LINT
VAR_INPUT
	divisor:LINT;
END_VAR

// Implicitly generated code : Only an Implementation suggestion
{noflow}
IF divisor = 0 THEN
	CheckDivLInt:=1;
ELSE
	CheckDivLInt:=divisor;
END_IF;
{flow}

END_FUNCTION

// ---- Checks/CheckDivLReal.TcPOU
// Implicitly generated code : DO NOT EDIT
FUNCTION CheckDivLReal : LREAL
VAR_INPUT
	divisor:LREAL;
END_VAR

// Implicitly generated code : Only an Implementation suggestion
{noflow}
IF divisor = 0 THEN
	CheckDivLReal:=1;
ELSE
	CheckDivLReal:=divisor;
END_IF;
{flow}

END_FUNCTION

// ---- Checks/CheckDivReal.TcPOU
// Implicitly generated code : DO NOT EDIT
FUNCTION CheckDivReal : REAL
VAR_INPUT
	divisor:REAL;
END_VAR

// Implicitly generated code : Only an Implementation suggestion
{noflow}
IF divisor = 0 THEN
	CheckDivReal:=1;
ELSE
	CheckDivReal:=divisor;
END_IF;
{flow}

END_FUNCTION

// ---- Checks/CheckLRangeSigned.TcPOU
// Implicitly generated code : DO NOT EDIT
FUNCTION CheckLRangeSigned : LINT
VAR_INPUT
	value, lower, upper: LINT;
END_VAR

// Implicitly generated code : Only an Implementation suggestion
{noflow}
IF (value < lower) THEN
	CheckLRangeSigned := lower;
ELSIF(value > upper) THEN
	CheckLRangeSigned := upper;
ELSE
	CheckLRangeSigned := value;
END_IF

{flow}

END_FUNCTION

// ---- Checks/CheckLRangeUnsigned.TcPOU
// Implicitly generated code : DO NOT EDIT
FUNCTION CheckLRangeUnsigned : ULINT
VAR_INPUT
	value, lower, upper: ULINT;
END_VAR

// Implicitly generated code : Only an Implementation suggestion
{noflow}
IF (value < lower) THEN
	CheckLRangeUnsigned := lower;
ELSIF(value > upper) THEN
	CheckLRangeUnsigned := upper;
ELSE
	CheckLRangeUnsigned := value;
END_IF
{flow}

END_FUNCTION

// ---- Checks/CheckPointer.TcPOU
// Implicitly generated code : DO NOT EDIT
FUNCTION CheckPointer : POINTER TO BYTE
VAR_INPUT 
	ptToTest : POINTER TO BYTE; // Destination address of the pointer
	iSize : DINT;		        // Size of the type the pointer points to. (e.g: 20 for POINTER TO ARRAY [0..9] OF INT) 
	iGran : DINT;		        // Granularity of the pointer access. This is the size of the biggest non-structured data type in the type the pointer points to. (e.g: 2 for POINTER TO ARRAY [0..9] OF INT)
	bWrite: BOOL;		        // Indicates read or write Access. TRUE = write access.
END_VAR

// Implicitly generated code : Only an Implementation suggestion
{noflow}
IF ptToTest=0 THEN
    ADSLOGSTR(ADSLOG_MSGTYPE_ERROR OR ADSLOG_MSGTYPE_STRING,'CheckPointer failed due to invalid address.','');
ELSIF iSize<=0 THEN
    ADSLOGSTR(ADSLOG_MSGTYPE_ERROR OR ADSLOG_MSGTYPE_STRING,'CheckPointer failed due to invalid size.','');
ELSIF iGran<=0 THEN
    ADSLOGSTR(ADSLOG_MSGTYPE_ERROR OR ADSLOG_MSGTYPE_STRING,'CheckPointer failed due to invalid granularity.','');
// -> Please note that the following memory area check is time consuming:
//ELSIF F_CheckMemoryArea(pData:=ptToTest,nSize:=DINT_TO_UDINT(iSize)) = E_TcMemoryArea.Unknown THEN
//    ADSLOGSTR(ADSLOG_MSGTYPE_ERROR OR ADSLOG_MSGTYPE_STRING,'CheckPointer failed due to unknown memory area.','');
END_IF
CheckPointer := ptToTest;
{flow}

END_FUNCTION

// ---- Checks/CheckRangeSigned.TcPOU
// Implicitly generated code : DO NOT EDIT
FUNCTION CheckRangeSigned : DINT
VAR_INPUT
	value, lower, upper: DINT;
END_VAR

// Implicitly generated code : Only an Implementation suggestion
{noflow}
IF (value < lower) THEN
	CheckRangeSigned := lower;
ELSIF(value > upper) THEN
	CheckRangeSigned := upper;
ELSE
	CheckRangeSigned := value;
END_IF
{flow}

END_FUNCTION

// ---- Checks/CheckRangeUnsigned.TcPOU
// Implicitly generated code : DO NOT EDIT
FUNCTION CheckRangeUnsigned : UDINT
VAR_INPUT
	value, lower, upper: UDINT;
END_VAR

// Implicitly generated code : Only an Implementation suggestion
{noflow}
IF (value < lower) THEN
	CheckRangeUnsigned := lower;
ELSIF(value > upper) THEN
	CheckRangeUnsigned := upper;
ELSE
	CheckRangeUnsigned := value;
END_IF
{flow}

END_FUNCTION

// ---- Functions/UpdateTimeStamp.TcPOU
FUNCTION UpdateTimeStamp 
VAR_INPUT
	stUser : REFERENCE TO ST_USER;
END_VAR
VAR
	fbGETSYSTEMTIME : GETSYSTEMTIME;
	
	stFileTime : T_FILETIME;
END_VAR


fbGETSYSTEMTIME(timeLoDW =>stFileTime.dwLowDateTime ,
				timeHiDW =>stFileTime.dwHighDateTime );
				
stUser.dtTIME_STAMP:= FILETIME_TO_DT(fileTime := stFileTime);

END_FUNCTION

// ---- POUs/FB_ERROR_CODE.TcPOU
FUNCTION_BLOCK FB_ERROR_CODE
VAR_INPUT
END_VAR
VAR_OUTPUT
END_VAR
VAR
END_VAR

END_FUNCTION_BLOCK

// ---- POUs/PISTONS_CYCLE.TcPOU
PROGRAM PISTONS_CYCLE
VAR
	
	bSTARTUP: BOOL:=FALSE;
	counter: INT;
	MANUALcOUNTER:int:=0;
	timimg: REAL:=0.2;
	bTestOpen:BOOL:=TRUE;
	bTestClose:BOOL:=TRUE;
END_VAR

IF NOT bSTARTUP THEN
	
	stPISTON_PARAM[1].nNAME:='FEEDER PUSHER';
	stPISTON_PARAM[1].bOPEN_BY_DEFAULT:=FALSE;
	stPISTON_PARAM[1].openTime:=timimg;
	stPISTON_PARAM[1].closeTime:=timimg;
	stPISTON_PARAM[1].timeoutOpen:=T#3S;
	stPISTON_PARAM[1].timeoutClose:=T#3S;
	stPISTON_PARAM[1].ePISTON_TYPE:= 0;
	
	
	stPISTON_PARAM[2].nNAME:='FEEDER HOLDER';
	stPISTON_PARAM[2].bOPEN_BY_DEFAULT:=FALSE;
	stPISTON_PARAM[2].openTime:=timimg;
	stPISTON_PARAM[2].closeTime:=timimg;
	stPISTON_PARAM[2].timeoutOpen:=T#2S;
	stPISTON_PARAM[2].timeoutClose:=T#2S;
	stPISTON_PARAM[2].ePISTON_TYPE:= 0;
	
	stPISTON_PARAM[15].nNAME:='FEEDER OPENER';
	stPISTON_PARAM[15].bOPEN_BY_DEFAULT:=FALSE;
	stPISTON_PARAM[15].openTime:=timimg;
	stPISTON_PARAM[15].closeTime:=timimg;
	stPISTON_PARAM[15].timeoutOpen:=T#2S;
	stPISTON_PARAM[15].timeoutClose:=T#2S;
	stPISTON_PARAM[15].ePISTON_TYPE:= 0;
	
	stPISTON_PARAM[3].nNAME:='SEPARATE1 LIFT';
	stPISTON_PARAM[3].bOPEN_BY_DEFAULT:=FALSE;
	stPISTON_PARAM[3].openTime:=timimg;
	stPISTON_PARAM[3].closeTime:=timimg;
	stPISTON_PARAM[3].timeoutOpen:=T#3S;
	stPISTON_PARAM[3].timeoutClose:=T#3S;
	stPISTON_PARAM[3].ePISTON_TYPE:= 0;
	
	
	stPISTON_PARAM[4].nNAME:='SEPARATE1 COLET';
	stPISTON_PARAM[4].bOPEN_BY_DEFAULT:=FALSE;
	stPISTON_PARAM[4].openTime:=timimg;
	stPISTON_PARAM[4].closeTime:=timimg;
	stPISTON_PARAM[4].timeoutOpen:=T#3S;
	stPISTON_PARAM[4].timeoutClose:=T#3S;
	stPISTON_PARAM[4].ePISTON_TYPE:= 0;
	
	
	stPISTON_PARAM[5].nNAME:='SEPARATE1 PULL';
	stPISTON_PARAM[5].bOPEN_BY_DEFAULT:=FALSE;
	stPISTON_PARAM[5].openTime:=timimg;
	stPISTON_PARAM[5].closeTime:=timimg;
	stPISTON_PARAM[5].timeoutOpen:=T#3S;
	stPISTON_PARAM[5].timeoutClose:=T#3S;
	stPISTON_PARAM[5].ePISTON_TYPE:= 0;
	
	
	stPISTON_PARAM[6].nNAME:='SEPARATE1 TRAY';
	stPISTON_PARAM[6].bOPEN_BY_DEFAULT:=FALSE;
	stPISTON_PARAM[6].openTime:=timimg;
	stPISTON_PARAM[6].closeTime:=timimg;
	stPISTON_PARAM[6].timeoutOpen:=T#3S;
	stPISTON_PARAM[6].timeoutClose:=T#3S;
	stPISTON_PARAM[6].ePISTON_TYPE:= 0;
	
	
	stPISTON_PARAM[7].nNAME:='SEPARATE1 PUSH PINS';
	stPISTON_PARAM[7].bOPEN_BY_DEFAULT:=FALSE;
	stPISTON_PARAM[7].openTime:=timimg;
	stPISTON_PARAM[7].closeTime:=timimg;
	stPISTON_PARAM[7].timeoutOpen:=T#3S;
	stPISTON_PARAM[7].timeoutClose:=T#3S;
	stPISTON_PARAM[7].ePISTON_TYPE:= 0;
	
	stPISTON_PARAM[16].nNAME:='SEPARATE1 TRAY PUSHER';
	stPISTON_PARAM[16].bOPEN_BY_DEFAULT:=FALSE;
	stPISTON_PARAM[16].openTime:=timimg;
	stPISTON_PARAM[16].closeTime:=timimg;
	stPISTON_PARAM[16].timeoutOpen:=T#3S;
	stPISTON_PARAM[16].timeoutClose:=T#3S;
	stPISTON_PARAM[16].ePISTON_TYPE:= 0;
	
	stPISTON_PARAM[17].nNAME:='SEPARATE1 TRAY DOOR';
	stPISTON_PARAM[17].bOPEN_BY_DEFAULT:=FALSE;
	stPISTON_PARAM[17].openTime:=timimg;
	stPISTON_PARAM[17].closeTime:=timimg;
	stPISTON_PARAM[17].timeoutOpen:=T#3S;
	stPISTON_PARAM[17].timeoutClose:=T#3S;
	stPISTON_PARAM[17].ePISTON_TYPE:= 0;
	
	stPISTON_PARAM[8].nNAME:='SEPARATE2 LIFT';
	stPISTON_PARAM[8].bOPEN_BY_DEFAULT:=FALSE;
	stPISTON_PARAM[8].openTime:=timimg;
	stPISTON_PARAM[8].closeTime:=timimg;
	stPISTON_PARAM[8].timeoutOpen:=T#3S;
	stPISTON_PARAM[8].timeoutClose:=T#3S;
	stPISTON_PARAM[8].ePISTON_TYPE:= 0;
	
	
	stPISTON_PARAM[9].nNAME:='SEPARATE2 COLET';
	stPISTON_PARAM[9].bOPEN_BY_DEFAULT:=FALSE;
	stPISTON_PARAM[9].openTime:=timimg;
	stPISTON_PARAM[9].closeTime:=timimg;
	stPISTON_PARAM[9].timeoutOpen:=T#3S;
	stPISTON_PARAM[9].timeoutClose:=T#3S;
	stPISTON_PARAM[9].ePISTON_TYPE:= 0;
	
	
	stPISTON_PARAM[10].nNAME:='SEPARATE2 PULL';
	stPISTON_PARAM[10].bOPEN_BY_DEFAULT:=FALSE;
	stPISTON_PARAM[10].openTime:=timimg;
	stPISTON_PARAM[10].closeTime:=timimg;
	stPISTON_PARAM[10].timeoutOpen:=T#3S;
	stPISTON_PARAM[10].timeoutClose:=T#3S;
	stPISTON_PARAM[10].ePISTON_TYPE:= 0;
	
	
	stPISTON_PARAM[11].nNAME:='SEPARATE2 TRAY';
	stPISTON_PARAM[11].bOPEN_BY_DEFAULT:=FALSE;
	stPISTON_PARAM[11].openTime:=timimg;
	stPISTON_PARAM[11].closeTime:=timimg;
	stPISTON_PARAM[11].timeoutOpen:=T#3S;
	stPISTON_PARAM[11].timeoutClose:=T#3S;
	stPISTON_PARAM[11].ePISTON_TYPE:= 0;
	
	stPISTON_PARAM[12].nNAME:='SEPARATE2 PUSH PINS';
	stPISTON_PARAM[12].bOPEN_BY_DEFAULT:=FALSE;
	stPISTON_PARAM[12].openTime:=timimg;
	stPISTON_PARAM[12].closeTime:=timimg;
	stPISTON_PARAM[12].timeoutOpen:=T#3S;
	stPISTON_PARAM[12].timeoutClose:=T#3S;
	stPISTON_PARAM[12].ePISTON_TYPE:= 0;
	
	stPISTON_PARAM[18].nNAME:='SEPARATE2 TRAY PUSHER';
	stPISTON_PARAM[18].bOPEN_BY_DEFAULT:=FALSE;
	stPISTON_PARAM[18].openTime:=timimg;
	stPISTON_PARAM[18].closeTime:=timimg;
	stPISTON_PARAM[18].timeoutOpen:=T#3S;
	stPISTON_PARAM[18].timeoutClose:=T#3S;
	stPISTON_PARAM[18].ePISTON_TYPE:= 0;
	
	stPISTON_PARAM[19].nNAME:='SEPARATE2 TRAY DOOR';
	stPISTON_PARAM[19].bOPEN_BY_DEFAULT:=FALSE;
	stPISTON_PARAM[19].openTime:=timimg;
	stPISTON_PARAM[19].closeTime:=timimg;
	stPISTON_PARAM[19].timeoutOpen:=T#3S;
	stPISTON_PARAM[19].timeoutClose:=T#3S;
	stPISTON_PARAM[19].ePISTON_TYPE:= 0;
	
	stPISTON_PARAM[13].nNAME:='DISPOSE OPENER';
	stPISTON_PARAM[13].bOPEN_BY_DEFAULT:=FALSE;
	stPISTON_PARAM[13].openTime:=0.5;
	stPISTON_PARAM[13].closeTime:=0.5;
	stPISTON_PARAM[13].timeoutOpen:=T#3S;
	stPISTON_PARAM[13].timeoutClose:=T#3S;
	stPISTON_PARAM[13].ePISTON_TYPE:= 0;
	
	stPISTON_PARAM[14].nNAME:='CLEAN';
	stPISTON_PARAM[14].bOPEN_BY_DEFAULT:=FALSE;
	stPISTON_PARAM[14].openTime:=timimg;
	stPISTON_PARAM[14].closeTime:=timimg;
	stPISTON_PARAM[14].timeoutOpen:=T#3S;
	stPISTON_PARAM[14].timeoutClose:=T#3S;
	stPISTON_PARAM[14].ePISTON_TYPE:= 0;
	
	stPISTON_PARAM[20].nNAME:='EXTRA ';
	stPISTON_PARAM[20].bOPEN_BY_DEFAULT:=FALSE;
	stPISTON_PARAM[20].openTime:=timimg;
	stPISTON_PARAM[20].closeTime:=timimg;
	stPISTON_PARAM[20].timeoutOpen:=T#3S;
	stPISTON_PARAM[20].timeoutClose:=T#3S;
	stPISTON_PARAM[20].ePISTON_TYPE:= 0;
	
	stPISTON_PARAM[21].nNAME:='DROP PUSHER';
	stPISTON_PARAM[21].bOPEN_BY_DEFAULT:=FALSE;
	stPISTON_PARAM[21].openTime:=0.5;
	stPISTON_PARAM[21].closeTime:=0.5;
	stPISTON_PARAM[21].timeoutOpen:=T#3S;
	stPISTON_PARAM[21].timeoutClose:=T#3S;
	stPISTON_PARAM[21].ePISTON_TYPE:= 0;
	
	stPISTON_PARAM[22].nNAME:='DROP OPENER';
	stPISTON_PARAM[22].bOPEN_BY_DEFAULT:=FALSE;
	stPISTON_PARAM[22].openTime:=timimg;
	stPISTON_PARAM[22].closeTime:=timimg;
	stPISTON_PARAM[22].timeoutOpen:=T#3S;
	stPISTON_PARAM[22].timeoutClose:=T#3S;
	stPISTON_PARAM[22].ePISTON_TYPE:= 0;
	
	//FOR counter:=1 TO iNUMBER_OF_PISTONS BY 1 DO
		//fbPiston[counter](stPISTON:=stPISTON_PARAM[counter]);
	//END_FOR;
	
	bSTARTUP:=TRUE;
END_IF

MANUALcOUNTER:=0;
FOR counter:=1 TO iNUMBER_OF_PISTONS BY 1 DO
	//IF fbPiston[counter].bMANUAL THEN
	//	bManual_mode:=TRUE;
	//	manualCounter:= manualCounter+1;
//	END_IF
	//fbPiston[counter]();
END_FOR;

IF manualCounter = 0 THEN
	bManual_mode:=FALSE;
END_IF
//feeder();
//clean();
//dispose();
//feeder();
//drop();
//separate1();
//separate2();

ACTION clean:
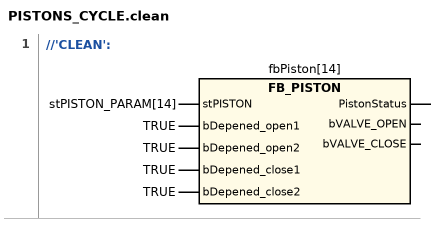
// NETWORK 1
// label: //'CLEAN'
fbPiston[14](
    stPISTON := stPISTON_PARAM[14],
    bDepened_open1 := TRUE,
    bDepened_open2 := TRUE,
    bDepened_close1 := TRUE,
    bDepened_close2 := TRUE); // FB_PISTON
END_ACTION

ACTION dispose:
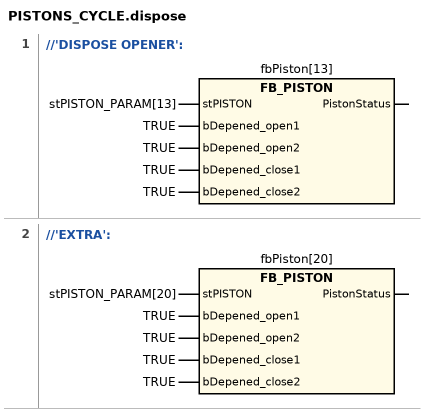
// NETWORK 1
// label: //'DISPOSE OPENER'
fbPiston[13](
    stPISTON := stPISTON_PARAM[13],
    bDepened_open1 := TRUE,
    bDepened_open2 := TRUE,
    bDepened_close1 := TRUE,
    bDepened_close2 := TRUE); // FB_PISTON

// NETWORK 2
// label: //'EXTRA'
fbPiston[20](
    stPISTON := stPISTON_PARAM[20],
    bDepened_open1 := TRUE,
    bDepened_open2 := TRUE,
    bDepened_close1 := TRUE,
    bDepened_close2 := TRUE); // FB_PISTON
END_ACTION

ACTION drop:
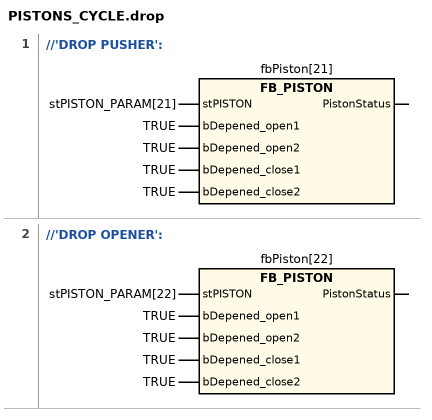
// NETWORK 1
// label: //'DROP PUSHER'
fbPiston[21](
    stPISTON := stPISTON_PARAM[21],
    bDepened_open1 := TRUE,
    bDepened_open2 := TRUE,
    bDepened_close1 := TRUE,
    bDepened_close2 := TRUE); // FB_PISTON

// NETWORK 2
// label: //'DROP OPENER'
fbPiston[22](
    stPISTON := stPISTON_PARAM[22],
    bDepened_open1 := TRUE,
    bDepened_open2 := TRUE,
    bDepened_close1 := TRUE,
    bDepened_close2 := TRUE); // FB_PISTON
END_ACTION

ACTION feeder:
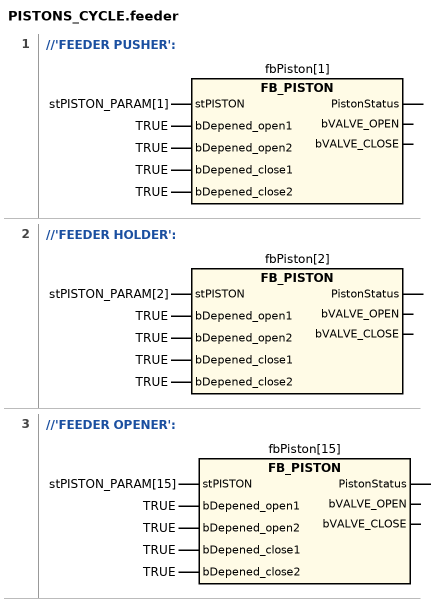
// NETWORK 1
// label: //'FEEDER PUSHER'
fbPiston[1](
    stPISTON := stPISTON_PARAM[1],
    bDepened_open1 := TRUE,
    bDepened_open2 := TRUE,
    bDepened_close1 := TRUE,
    bDepened_close2 := TRUE); // FB_PISTON

// NETWORK 2
// label: //'FEEDER HOLDER'
fbPiston[2](
    stPISTON := stPISTON_PARAM[2],
    bDepened_open1 := TRUE,
    bDepened_open2 := TRUE,
    bDepened_close1 := TRUE,
    bDepened_close2 := TRUE); // FB_PISTON

// NETWORK 3
// label: //'FEEDER OPENER'
fbPiston[15](
    stPISTON := stPISTON_PARAM[15],
    bDepened_open1 := TRUE,
    bDepened_open2 := TRUE,
    bDepened_close1 := TRUE,
    bDepened_close2 := TRUE); // FB_PISTON
END_ACTION

ACTION separate1:
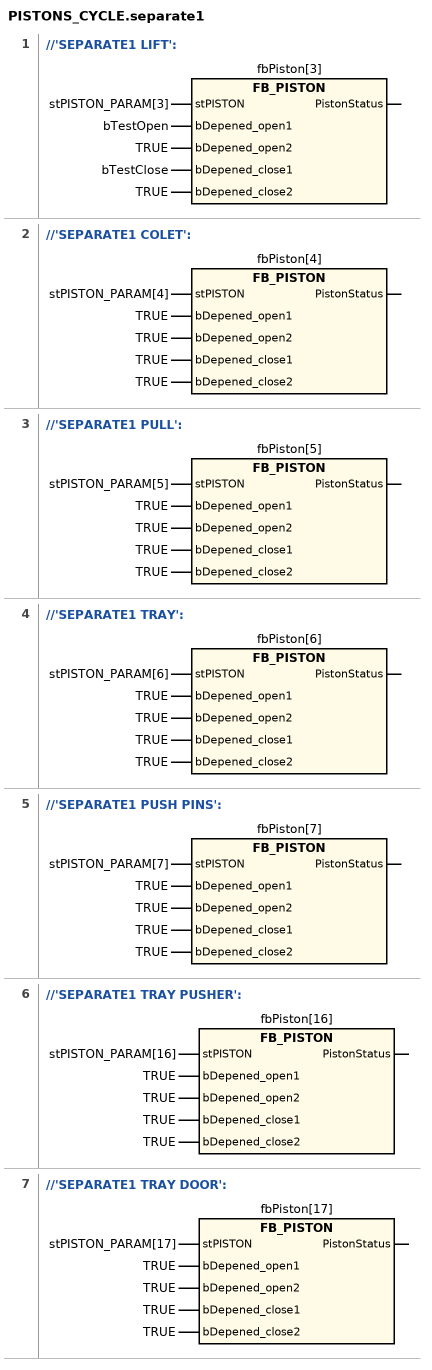
// NETWORK 1
// label: //'SEPARATE1 LIFT'
fbPiston[3](
    stPISTON := stPISTON_PARAM[3],
    bDepened_open1 := bTestOpen,
    bDepened_open2 := TRUE,
    bDepened_close1 := bTestClose,
    bDepened_close2 := TRUE); // FB_PISTON

// NETWORK 2
// label: //'SEPARATE1 COLET'
fbPiston[4](
    stPISTON := stPISTON_PARAM[4],
    bDepened_open1 := TRUE,
    bDepened_open2 := TRUE,
    bDepened_close1 := TRUE,
    bDepened_close2 := TRUE); // FB_PISTON

// NETWORK 3
// label: //'SEPARATE1 PULL'
fbPiston[5](
    stPISTON := stPISTON_PARAM[5],
    bDepened_open1 := TRUE,
    bDepened_open2 := TRUE,
    bDepened_close1 := TRUE,
    bDepened_close2 := TRUE); // FB_PISTON

// NETWORK 4
// label: //'SEPARATE1 TRAY'
fbPiston[6](
    stPISTON := stPISTON_PARAM[6],
    bDepened_open1 := TRUE,
    bDepened_open2 := TRUE,
    bDepened_close1 := TRUE,
    bDepened_close2 := TRUE); // FB_PISTON

// NETWORK 5
// label: //'SEPARATE1 PUSH PINS'
fbPiston[7](
    stPISTON := stPISTON_PARAM[7],
    bDepened_open1 := TRUE,
    bDepened_open2 := TRUE,
    bDepened_close1 := TRUE,
    bDepened_close2 := TRUE); // FB_PISTON

// NETWORK 6
// label: //'SEPARATE1 TRAY PUSHER'
fbPiston[16](
    stPISTON := stPISTON_PARAM[16],
    bDepened_open1 := TRUE,
    bDepened_open2 := TRUE,
    bDepened_close1 := TRUE,
    bDepened_close2 := TRUE); // FB_PISTON

// NETWORK 7
// label: //'SEPARATE1 TRAY DOOR'
fbPiston[17](
    stPISTON := stPISTON_PARAM[17],
    bDepened_open1 := TRUE,
    bDepened_open2 := TRUE,
    bDepened_close1 := TRUE,
    bDepened_close2 := TRUE); // FB_PISTON
END_ACTION

ACTION separate2:
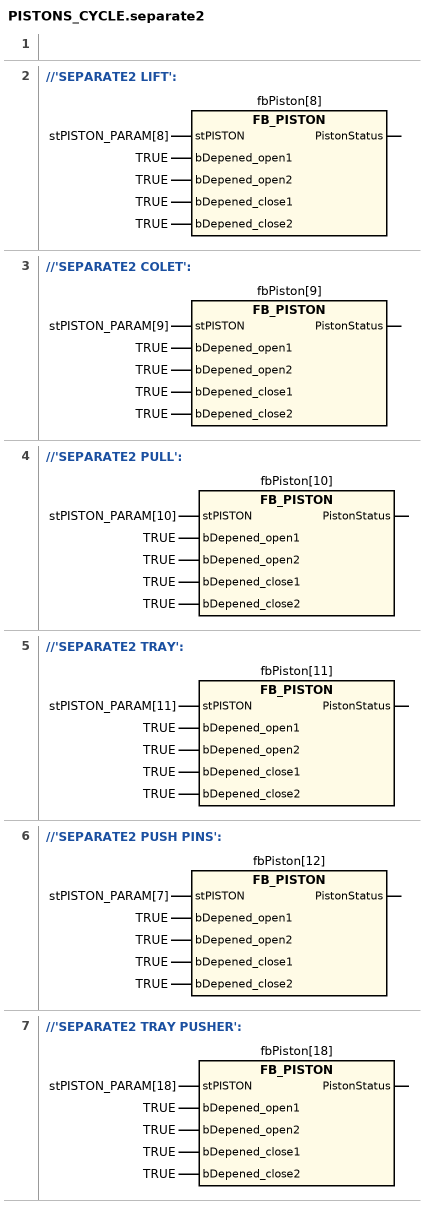
// NETWORK 1

// NETWORK 2
// label: //'SEPARATE2 LIFT'
fbPiston[8](
    stPISTON := stPISTON_PARAM[8],
    bDepened_open1 := TRUE,
    bDepened_open2 := TRUE,
    bDepened_close1 := TRUE,
    bDepened_close2 := TRUE); // FB_PISTON

